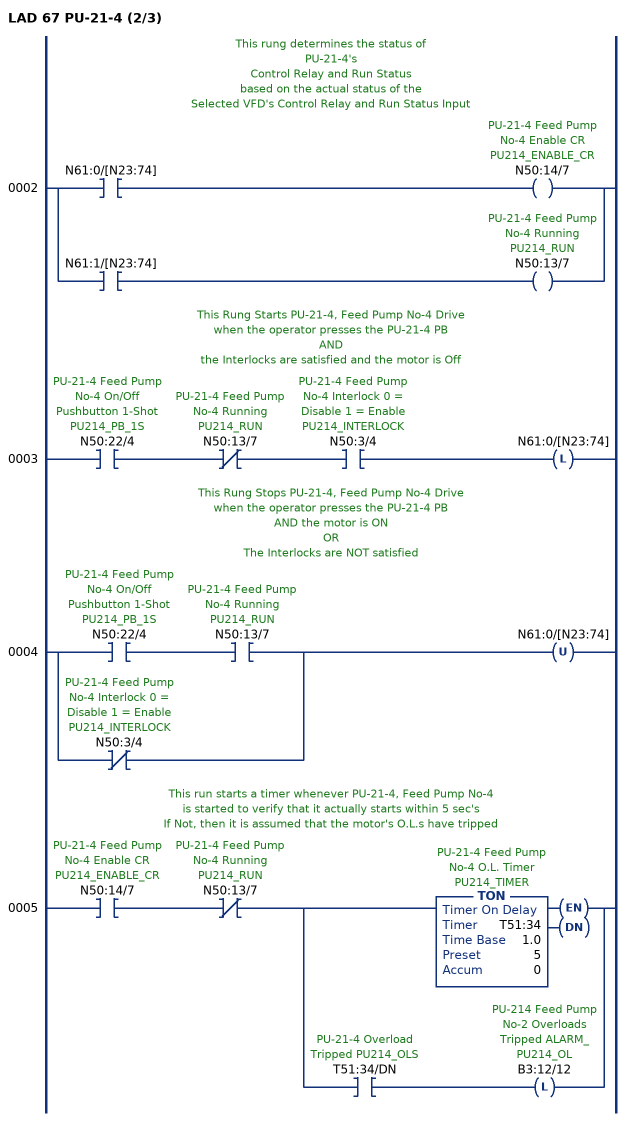
% Rung: 2 %
% This rung determines the status of
% PU-21-4's
% Control Relay and Run Status
% based on the actual status of the
% Selected VFD's Control Relay and Run Status Input %
SOR BST XIC N61:0/[N23:74] OTE N50:14/7 NXB XIC N61:1/[N23:74] OTE N50:13/7 BND EOR
%   N61:0  VFD_ENABLE_BITS  "These Bits Enable the appropriate VFD" %
%   N23:74  FIC214_OUT_PTR  "FIC-21-4 Feed Flow No-4 Output Pointer Determines which VFD is controled by FIC" %
%   N50:14/7  PU214_ENABLE_CR  "PU-21-4 Feed Pump No-4 Enable CR" %
%   N61:1  VFD_RUN_BITS_1  "These Bits Initcate the Status Off/Running for the appropriate VFD" %
%   N50:13/7  PU214_RUN  "PU-21-4 Feed Pump No-4 Running" %
% Rung: 3 %
% This Rung Starts PU-21-4, Feed Pump No-4 Drive
% when the operator presses the PU-21-4 PB
% AND
% the Interlocks are satisfied and the motor is Off %
SOR XIC N50:22/4 XIO N50:13/7 XIC N50:3/4 OTL N61:0/[N23:74] EOR
%   N50:22/4  PU214_PB_1S  "PU-21-4 Feed Pump No-4 On/Off Pushbutton 1-Shot" %
%   N50:13/7  PU214_RUN  "PU-21-4 Feed Pump No-4 Running" %
%   N50:3/4  PU214_INTERLOCK  "PU-21-4 Feed Pump No-4 Interlock 0 = Disable 1 = Enable" %
%   N61:0  VFD_ENABLE_BITS  "These Bits Enable the appropriate VFD" %
%   N23:74  FIC214_OUT_PTR  "FIC-21-4 Feed Flow No-4 Output Pointer Determines which VFD is controled by FIC" %
% Rung: 4 %
% This Rung Stops PU-21-4, Feed Pump No-4 Drive
% when the operator presses the PU-21-4 PB
% AND the motor is ON
% OR
% The Interlocks are NOT satisfied %
SOR BST XIC N50:22/4 XIC N50:13/7 NXB XIO N50:3/4 BND OTU N61:0/[N23:74] EOR
%   N50:22/4  PU214_PB_1S  "PU-21-4 Feed Pump No-4 On/Off Pushbutton 1-Shot" %
%   N50:13/7  PU214_RUN  "PU-21-4 Feed Pump No-4 Running" %
%   N50:3/4  PU214_INTERLOCK  "PU-21-4 Feed Pump No-4 Interlock 0 = Disable 1 = Enable" %
%   N61:0  VFD_ENABLE_BITS  "These Bits Enable the appropriate VFD" %
%   N23:74  FIC214_OUT_PTR  "FIC-21-4 Feed Flow No-4 Output Pointer Determines which VFD is controled by FIC" %
% Rung: 5 %
% This run starts a timer whenever PU-21-4, Feed Pump No-4
% is started to verify that it actually starts within 5 sec's
% If Not, then it is assumed that the motor's O.L.s have tripped %
SOR XIC N50:14/7 XIO N50:13/7 BST TON T51:34 1.0 5 0 NXB XIC T51:34/DN OTL B3:12/12 BND EOR
%   N50:14/7  PU214_ENABLE_CR  "PU-21-4 Feed Pump No-4 Enable CR" %
%   N50:13/7  PU214_RUN  "PU-21-4 Feed Pump No-4 Running" %
%   T51:34  PU214_TIMER  "PU-21-4 Feed Pump No-4 O.L. Timer" %
%   T51:34/DN  PU214_OLS  "PU-21-4 Overload Tripped" %
%   B3:12/12  ALARM_PU214_OL  "PU-214 Feed Pump No-2 Overloads Tripped" %

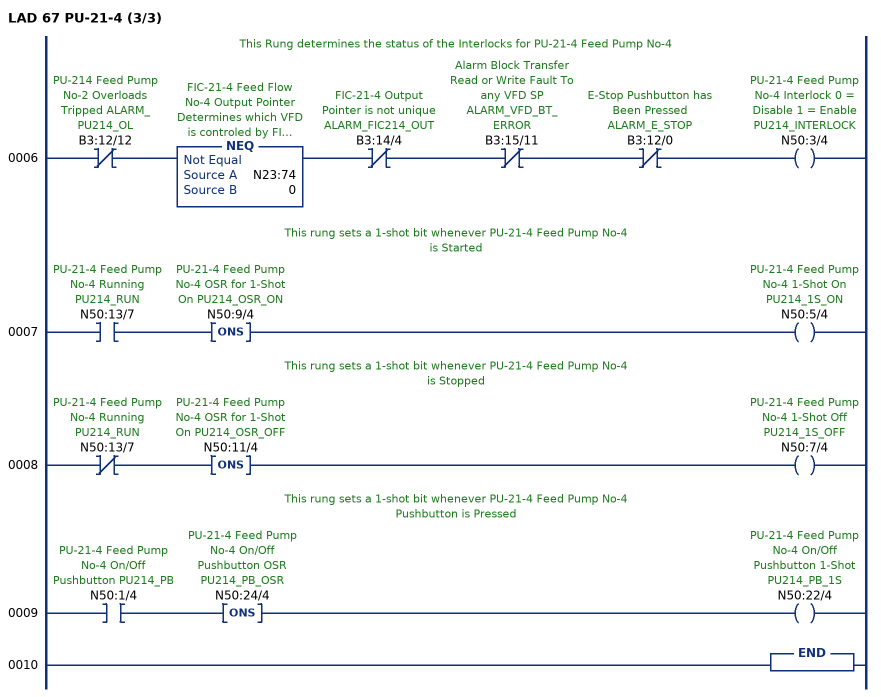
% Rung: 6 %
% This Rung determines the status of the Interlocks for PU-21-4 Feed Pump No-4 %
SOR XIO B3:12/12 NEQ N23:74 0 XIO B3:14/4 XIO B3:15/11 XIO B3:12/0 OTE N50:3/4 EOR
%   B3:12/12  ALARM_PU214_OL  "PU-214 Feed Pump No-2 Overloads Tripped" %
%   N23:74  FIC214_OUT_PTR  "FIC-21-4 Feed Flow No-4 Output Pointer Determines which VFD is controled by FIC" %
%   B3:14/4  ALARM_FIC214_OUT  "FIC-21-4 Output Pointer is not unique" %
%   B3:15/11  ALARM_VFD_BT_ERROR  "Alarm Block Transfer Read or Write Fault To any VFD SP" %
%   B3:12/0  ALARM_E_STOP  "E-Stop Pushbutton has Been Pressed" %
%   N50:3/4  PU214_INTERLOCK  "PU-21-4 Feed Pump No-4 Interlock 0 = Disable 1 = Enable" %
% Rung: 7 %
% This rung sets a 1-shot bit whenever PU-21-4 Feed Pump No-4
% is Started %
SOR XIC N50:13/7 OSR N50:9/4 OTE N50:5/4 EOR
%   N50:13/7  PU214_RUN  "PU-21-4 Feed Pump No-4 Running" %
%   N50:9/4  PU214_OSR_ON  "PU-21-4 Feed Pump No-4 OSR for 1-Shot On" %
%   N50:5/4  PU214_1S_ON  "PU-21-4 Feed Pump No-4 1-Shot On" %
% Rung: 8 %
% This rung sets a 1-shot bit whenever PU-21-4 Feed Pump No-4
% is Stopped %
SOR XIO N50:13/7 OSR N50:11/4 OTE N50:7/4 EOR
%   N50:13/7  PU214_RUN  "PU-21-4 Feed Pump No-4 Running" %
%   N50:11/4  PU214_OSR_OFF  "PU-21-4 Feed Pump No-4 OSR for 1-Shot On" %
%   N50:7/4  PU214_1S_OFF  "PU-21-4 Feed Pump No-4 1-Shot Off" %
% Rung: 9 %
% This rung sets a 1-shot bit whenever PU-21-4 Feed Pump No-4
% Pushbutton is Pressed %
SOR XIC N50:1/4 OSR N50:24/4 OTE N50:22/4 EOR
%   N50:1/4  PU214_PB  "PU-21-4 Feed Pump No-4 On/Off Pushbutton" %
%   N50:24/4  PU214_PB_OSR  "PU-21-4 Feed Pump No-4 On/Off Pushbutton OSR" %
%   N50:22/4  PU214_PB_1S  "PU-21-4 Feed Pump No-4 On/Off Pushbutton 1-Shot" %
% Rung: 10 %
SOR END EOR

LADDER 69 "PU-22-1"    % PU-22-1 Level Pump No-1 Controls %
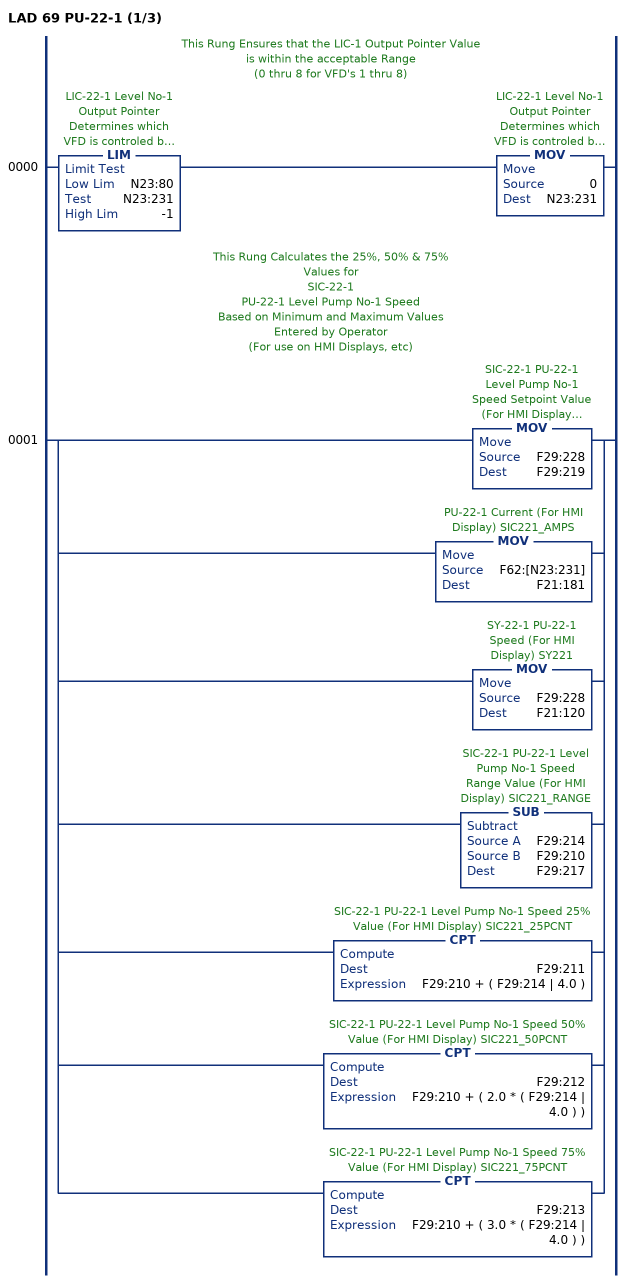
% Rung: 0 %
% This Rung Ensures that the LIC-1 Output Pointer Value
% is within the acceptable Range
% (0 thru 8 for VFD's 1 thru 8) %
SOR LIM N23:80 N23:231 -1 MOV 0 N23:231 EOR
%   N23:80  MAX_VFD_ALLOWED_1  "Maximum Number of VFDs Available Plus 1" %
%   N23:231  LIC221_OUT_PTR  "LIC-22-1 Level No-1 Output Pointer Determines which VFD is controled by LIC" %
% Rung: 1 %
% This Rung Calculates the 25%, 50% & 75%
% Values for
% SIC-22-1
% PU-22-1 Level Pump No-1 Speed
% Based on Minimum and Maximum Values
% Entered by Operator
% (For use on HMI Displays, etc) %
SOR BST MOV F29:228 F29:219 NXB MOV F62:[N23:231] F21:181 NXB MOV F29:228 F21:120 NXB SUB F29:214 F29:210 F29:217 NXB CPT F29:211 " F29:210 + ( F29:214 | 4.0 ) " NXB CPT F29:212 " F29:210 + ( 2.0 * ( F29:214 | 4.0 ) ) " NXB CPT F29:213 " F29:210 + ( 3.0 * ( F29:214 | 4.0 ) ) " BND EOR
%   F29:228  LIC221_OUT_FP  "LIC-22-1 Output Value (For HMI Display)" %
%   F29:219  SIC221_SP_FP  "SIC-22-1 PU-22-1 Level Pump No-1 Speed Setpoint Value (For HMI Display)" %
%   N23:231  LIC221_OUT_PTR  "LIC-22-1 Level No-1 Output Pointer Determines which VFD is controled by LIC" %
%   F21:181  SIC221_AMPS  "PU-22-1 Current (For HMI Display)" %
%   F21:120  SY221  "SY-22-1 PU-22-1 Speed (For HMI Display)" %
%   F29:214  SIC221_MAX  "SIC-22-1 PU-22-1 Level Pump No-1 Freq at 100% Value (For HMI Display)" %
%   F29:210  SIC221_MIN  "SIC-22-1 PU-22-1 Level Pump No-1 Speed 0% Value (For HMI Display)" %
%   F29:217  SIC221_RANGE  "SIC-22-1 PU-22-1 Level Pump No-1 Speed Range Value (For HMI Display)" %
%   F29:211  SIC221_25PCNT  "SIC-22-1 PU-22-1 Level Pump No-1 Speed 25% Value (For HMI Display)" %
%   F29:212  SIC221_50PCNT  "SIC-22-1 PU-22-1 Level Pump No-1 Speed 50% Value (For HMI Display)" %
%   F29:213  SIC221_75PCNT  "SIC-22-1 PU-22-1 Level Pump No-1 Speed 75% Value (For HMI Display)" %

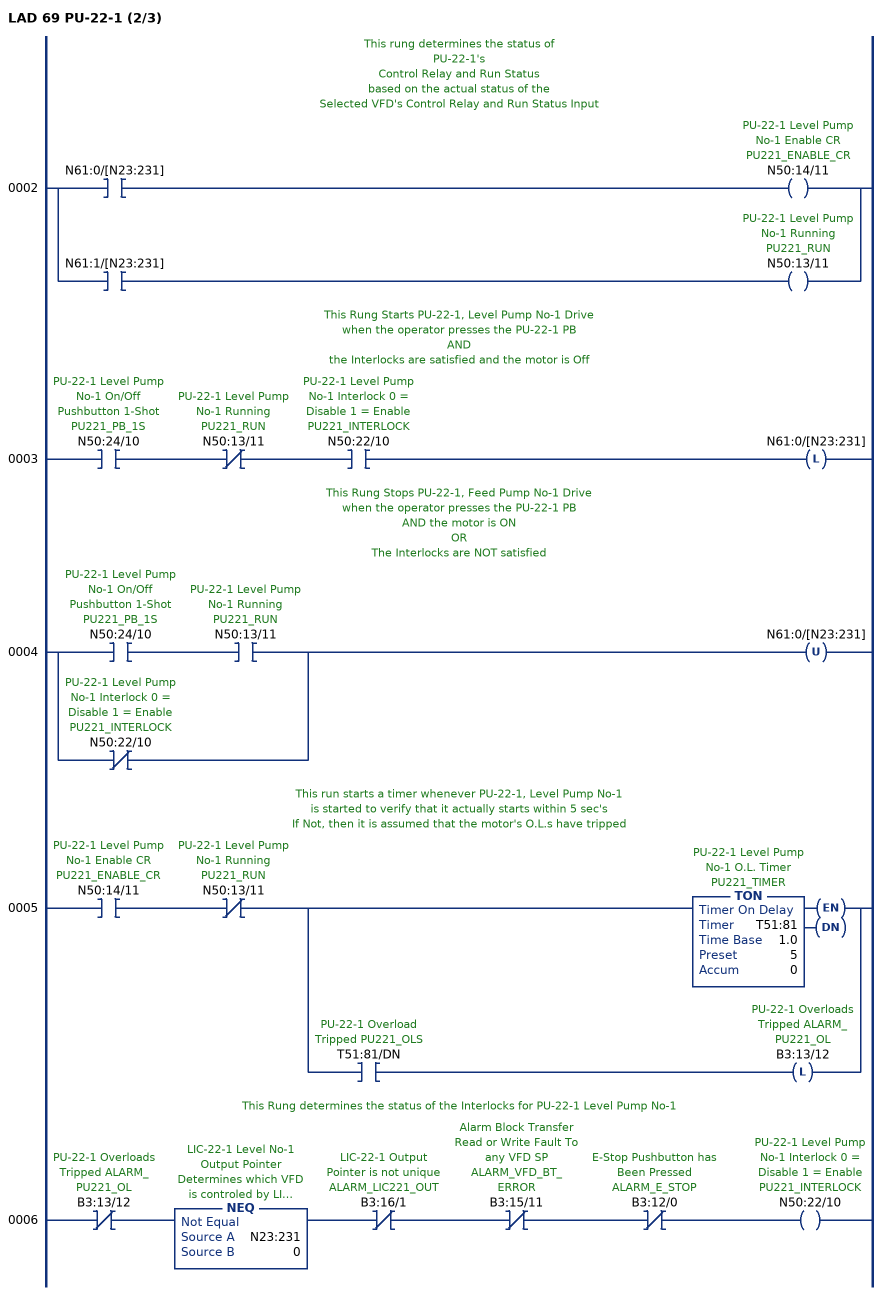
% Rung: 2 %
% This rung determines the status of
% PU-22-1's
% Control Relay and Run Status
% based on the actual status of the
% Selected VFD's Control Relay and Run Status Input %
SOR BST XIC N61:0/[N23:231] OTE N50:14/11 NXB XIC N61:1/[N23:231] OTE N50:13/11 BND EOR
%   N61:0  VFD_ENABLE_BITS  "These Bits Enable the appropriate VFD" %
%   N23:231  LIC221_OUT_PTR  "LIC-22-1 Level No-1 Output Pointer Determines which VFD is controled by LIC" %
%   N50:14/11  PU221_ENABLE_CR  "PU-22-1 Level Pump No-1 Enable CR" %
%   N61:1  VFD_RUN_BITS_1  "These Bits Initcate the Status Off/Running for the appropriate VFD" %
%   N50:13/11  PU221_RUN  "PU-22-1 Level Pump No-1 Running" %
% Rung: 3 %
% This Rung Starts PU-22-1, Level Pump No-1 Drive
% when the operator presses the PU-22-1 PB
% AND
% the Interlocks are satisfied and the motor is Off %
SOR XIC N50:24/10 XIO N50:13/11 XIC N50:22/10 OTL N61:0/[N23:231] EOR
%   N50:24/10  PU221_PB_1S  "PU-22-1 Level Pump No-1 On/Off Pushbutton 1-Shot" %
%   N50:13/11  PU221_RUN  "PU-22-1 Level Pump No-1 Running" %
%   N50:22/10  PU221_INTERLOCK  "PU-22-1 Level Pump No-1 Interlock 0 = Disable 1 = Enable" %
%   N61:0  VFD_ENABLE_BITS  "These Bits Enable the appropriate VFD" %
%   N23:231  LIC221_OUT_PTR  "LIC-22-1 Level No-1 Output Pointer Determines which VFD is controled by LIC" %
% Rung: 4 %
% This Rung Stops PU-22-1, Feed Pump No-1 Drive
% when the operator presses the PU-22-1 PB
% AND the motor is ON
% OR
% The Interlocks are NOT satisfied %
SOR BST XIC N50:24/10 XIC N50:13/11 NXB XIO N50:22/10 BND OTU N61:0/[N23:231] EOR
%   N50:24/10  PU221_PB_1S  "PU-22-1 Level Pump No-1 On/Off Pushbutton 1-Shot" %
%   N50:13/11  PU221_RUN  "PU-22-1 Level Pump No-1 Running" %
%   N50:22/10  PU221_INTERLOCK  "PU-22-1 Level Pump No-1 Interlock 0 = Disable 1 = Enable" %
%   N61:0  VFD_ENABLE_BITS  "These Bits Enable the appropriate VFD" %
%   N23:231  LIC221_OUT_PTR  "LIC-22-1 Level No-1 Output Pointer Determines which VFD is controled by LIC" %
% Rung: 5 %
% This run starts a timer whenever PU-22-1, Level Pump No-1
% is started to verify that it actually starts within 5 sec's
% If Not, then it is assumed that the motor's O.L.s have tripped %
SOR XIC N50:14/11 XIO N50:13/11 BST TON T51:81 1.0 5 0 NXB XIC T51:81/DN OTL B3:13/12 BND EOR
%   N50:14/11  PU221_ENABLE_CR  "PU-22-1 Level Pump No-1 Enable CR" %
%   N50:13/11  PU221_RUN  "PU-22-1 Level Pump No-1 Running" %
%   T51:81  PU221_TIMER  "PU-22-1 Level Pump No-1 O.L. Timer" %
%   T51:81/DN  PU221_OLS  "PU-22-1 Overload Tripped" %
%   B3:13/12  ALARM_PU221_OL  "PU-22-1 Overloads Tripped" %
% Rung: 6 %
% This Rung determines the status of the Interlocks for PU-22-1 Level Pump No-1 %
SOR XIO B3:13/12 NEQ N23:231 0 XIO B3:16/1 XIO B3:15/11 XIO B3:12/0 OTE N50:22/10 EOR
%   B3:13/12  ALARM_PU221_OL  "PU-22-1 Overloads Tripped" %
%   N23:231  LIC221_OUT_PTR  "LIC-22-1 Level No-1 Output Pointer Determines which VFD is controled by LIC" %
%   B3:16/1  ALARM_LIC221_OUT  "LIC-22-1 Output Pointer is not unique" %
%   B3:15/11  ALARM_VFD_BT_ERROR  "Alarm Block Transfer Read or Write Fault To any VFD SP" %
%   B3:12/0  ALARM_E_STOP  "E-Stop Pushbutton has Been Pressed" %
%   N50:22/10  PU221_INTERLOCK  "PU-22-1 Level Pump No-1 Interlock 0 = Disable 1 = Enable" %

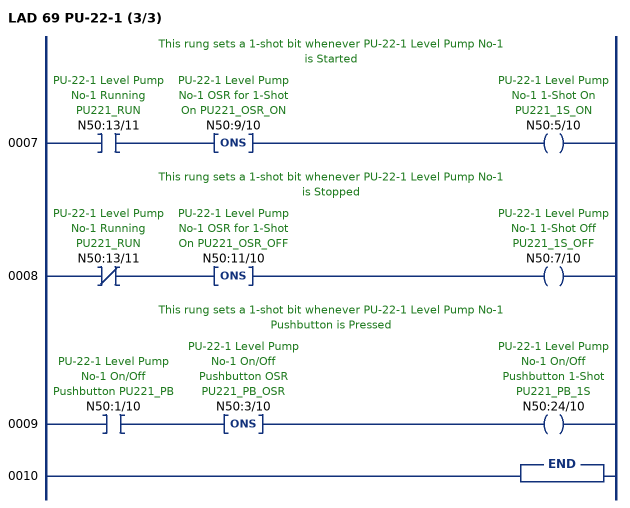
% Rung: 7 %
% This rung sets a 1-shot bit whenever PU-22-1 Level Pump No-1
% is Started %
SOR XIC N50:13/11 OSR N50:9/10 OTE N50:5/10 EOR
%   N50:13/11  PU221_RUN  "PU-22-1 Level Pump No-1 Running" %
%   N50:9/10  PU221_OSR_ON  "PU-22-1 Level Pump No-1 OSR for 1-Shot On" %
%   N50:5/10  PU221_1S_ON  "PU-22-1 Level Pump No-1 1-Shot On" %
% Rung: 8 %
% This rung sets a 1-shot bit whenever PU-22-1 Level Pump No-1
% is Stopped %
SOR XIO N50:13/11 OSR N50:11/10 OTE N50:7/10 EOR
%   N50:13/11  PU221_RUN  "PU-22-1 Level Pump No-1 Running" %
%   N50:11/10  PU221_OSR_OFF  "PU-22-1 Level Pump No-1 OSR for 1-Shot On" %
%   N50:7/10  PU221_1S_OFF  "PU-22-1 Level Pump No-1 1-Shot Off" %
% Rung: 9 %
% This rung sets a 1-shot bit whenever PU-22-1 Level Pump No-1
% Pushbutton is Pressed %
SOR XIC N50:1/10 OSR N50:3/10 OTE N50:24/10 EOR
%   N50:1/10  PU221_PB  "PU-22-1 Level Pump No-1 On/Off Pushbutton" %
%   N50:3/10  PU221_PB_OSR  "PU-22-1 Level Pump No-1 On/Off Pushbutton OSR" %
%   N50:24/10  PU221_PB_1S  "PU-22-1 Level Pump No-1 On/Off Pushbutton 1-Shot" %
% Rung: 10 %
SOR END EOR

LADDER 71 "PU-23"    % PU-23 Hot Oil Circ Pump Controls %
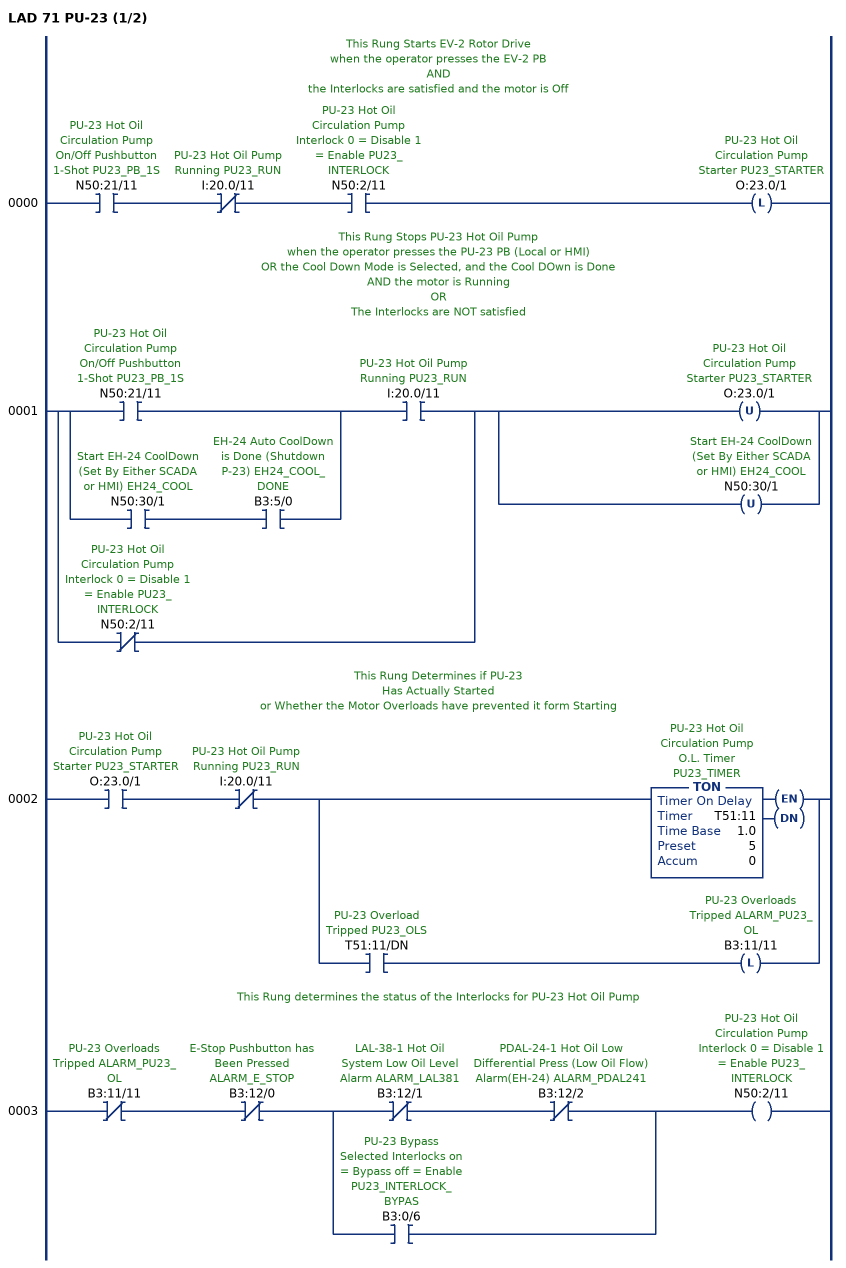
% Rung: 0 %
% This Rung Starts EV-2 Rotor Drive
% when the operator presses the EV-2 PB
% AND
% the Interlocks are satisfied and the motor is Off %
SOR XIC N50:21/11 XIO I:20.0/11 XIC N50:2/11 OTL O:23.0/1 EOR
%   N50:21/11  PU23_PB_1S  "PU-23 Hot Oil Circulation Pump On/Off Pushbutton 1-Shot" %
%   I:20.0/11  PU23_RUN  "PU-23 Hot Oil Pump Running" %
%   N50:2/11  PU23_INTERLOCK  "PU-23 Hot Oil Circulation Pump Interlock 0 = Disable 1 = Enable" %
%   O:23.0/1  PU23_STARTER  "PU-23 Hot Oil Circulation Pump Starter" %
% Rung: 1 %
% This Rung Stops PU-23 Hot Oil Pump
% when the operator presses the PU-23 PB (Local or HMI)
% OR the Cool Down Mode is Selected, and the Cool DOwn is Done
% AND the motor is Running
% OR
% The Interlocks are NOT satisfied %
SOR BST BST XIC N50:21/11 NXB XIC N50:30/1 XIC B3:5/0 BND XIC I:20.0/11 NXB XIO N50:2/11 BND BST OTU O:23.0/1 NXB OTU N50:30/1 BND EOR
%   N50:21/11  PU23_PB_1S  "PU-23 Hot Oil Circulation Pump On/Off Pushbutton 1-Shot" %
%   N50:30/1  EH24_COOL  "Start EH-24 CoolDown (Set By Either SCADA or HMI)" %
%   B3:5/0  EH24_COOL_DONE  "EH-24 Auto CoolDown is Done (Shutdown P-23)" %
%   I:20.0/11  PU23_RUN  "PU-23 Hot Oil Pump Running" %
%   N50:2/11  PU23_INTERLOCK  "PU-23 Hot Oil Circulation Pump Interlock 0 = Disable 1 = Enable" %
%   O:23.0/1  PU23_STARTER  "PU-23 Hot Oil Circulation Pump Starter" %
% Rung: 2 %
% This Rung Determines if PU-23
% Has Actually Started
% or Whether the Motor Overloads have prevented it form Starting %
SOR XIC O:23.0/1 XIO I:20.0/11 BST TON T51:11 1.0 5 0 NXB XIC T51:11/DN OTL B3:11/11 BND EOR
%   O:23.0/1  PU23_STARTER  "PU-23 Hot Oil Circulation Pump Starter" %
%   I:20.0/11  PU23_RUN  "PU-23 Hot Oil Pump Running" %
%   T51:11  PU23_TIMER  "PU-23 Hot Oil Circulation Pump O.L. Timer" %
%   T51:11/DN  PU23_OLS  "PU-23 Overload Tripped" %
%   B3:11/11  ALARM_PU23_OL  "PU-23 Overloads Tripped" %
% Rung: 3 %
% This Rung determines the status of the Interlocks for PU-23 Hot Oil Pump %
SOR XIO B3:11/11 XIO B3:12/0 BST XIO B3:12/1 XIO B3:12/2 NXB XIC B3:0/6 BND OTE N50:2/11 EOR
%   B3:11/11  ALARM_PU23_OL  "PU-23 Overloads Tripped" %
%   B3:12/0  ALARM_E_STOP  "E-Stop Pushbutton has Been Pressed" %
%   B3:12/1  ALARM_LAL381  "LAL-38-1 Hot Oil System Low Oil Level Alarm" %
%   B3:12/2  ALARM_PDAL241  "PDAL-24-1 Hot Oil Low Differential Press (Low Oil Flow) Alarm(EH-24)" %
%   B3:0/6  PU23_INTERLOCK_BYPAS  "PU-23 Bypass Selected Interlocks on = Bypass off = Enable" %
%   N50:2/11  PU23_INTERLOCK  "PU-23 Hot Oil Circulation Pump Interlock 0 = Disable 1 = Enable" %

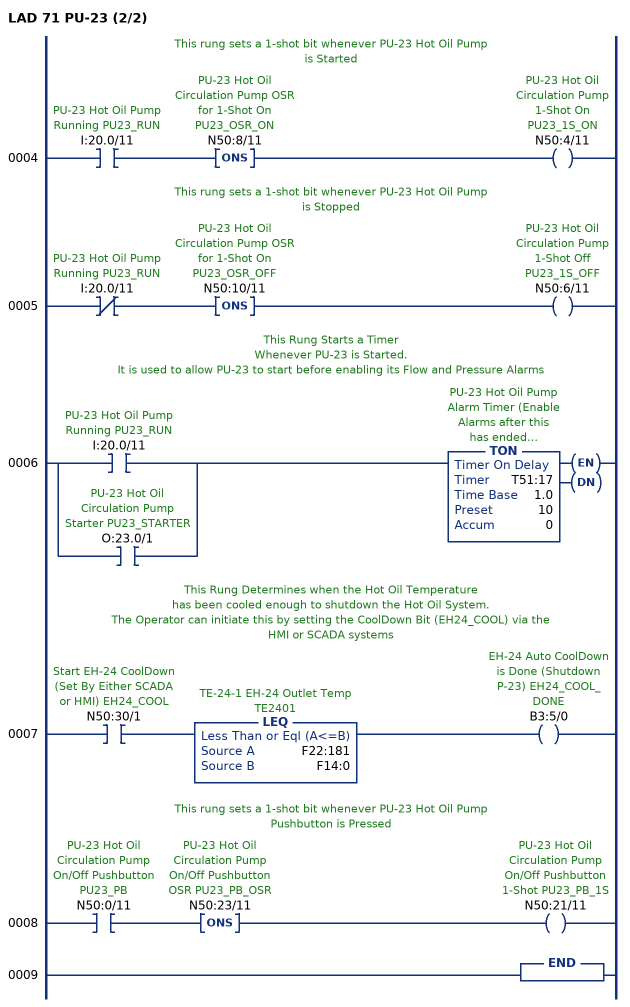
% Rung: 4 %
% This rung sets a 1-shot bit whenever PU-23 Hot Oil Pump
% is Started %
SOR XIC I:20.0/11 OSR N50:8/11 OTE N50:4/11 EOR
%   I:20.0/11  PU23_RUN  "PU-23 Hot Oil Pump Running" %
%   N50:8/11  PU23_OSR_ON  "PU-23 Hot Oil Circulation Pump OSR for 1-Shot On" %
%   N50:4/11  PU23_1S_ON  "PU-23 Hot Oil Circulation Pump 1-Shot On" %
% Rung: 5 %
% This rung sets a 1-shot bit whenever PU-23 Hot Oil Pump
% is Stopped %
SOR XIO I:20.0/11 OSR N50:10/11 OTE N50:6/11 EOR
%   I:20.0/11  PU23_RUN  "PU-23 Hot Oil Pump Running" %
%   N50:10/11  PU23_OSR_OFF  "PU-23 Hot Oil Circulation Pump OSR for 1-Shot On" %
%   N50:6/11  PU23_1S_OFF  "PU-23 Hot Oil Circulation Pump 1-Shot Off" %
% Rung: 6 %
% This Rung Starts a Timer
% Whenever PU-23 is Started.
% It is used to allow PU-23 to start before enabling its Flow and Pressure Alarms %
SOR BST XIC I:20.0/11 NXB XIC O:23.0/1 BND TON T51:17 1.0 10 0 EOR
%   I:20.0/11  PU23_RUN  "PU-23 Hot Oil Pump Running" %
%   O:23.0/1  PU23_STARTER  "PU-23 Hot Oil Circulation Pump Starter" %
%   T51:17  PU23_ALARM_TMR  "PU-23 Hot Oil Pump Alarm Timer (Enable Alarms after this has ended)" %
% Rung: 7 %
% This Rung Determines when the Hot Oil Temperature
% has been cooled enough to shutdown the Hot Oil System.
% The Operator can initiate this by setting the CoolDown Bit (EH24_COOL) via the
% HMI or SCADA systems %
SOR XIC N50:30/1 LEQ F22:181 F14:0 OTE B3:5/0 EOR
%   N50:30/1  EH24_COOL  "Start EH-24 CoolDown (Set By Either SCADA or HMI)" %
%   F22:181  TE2401  "TE-24-1 EH-24 Outlet Temp" %
%   F14:0  EH24_COOLDOWN_SP  "EH-24 CoolDown Setpoint" %
%   B3:5/0  EH24_COOL_DONE  "EH-24 Auto CoolDown is Done (Shutdown P-23)" %
% Rung: 8 %
% This rung sets a 1-shot bit whenever PU-23 Hot Oil Pump
% Pushbutton is Pressed %
SOR XIC N50:0/11 OSR N50:23/11 OTE N50:21/11 EOR
%   N50:0/11  PU23_PB  "PU-23 Hot Oil Circulation Pump On/Off Pushbutton" %
%   N50:23/11  PU23_PB_OSR  "PU-23 Hot Oil Circulation Pump On/Off Pushbutton OSR" %
%   N50:21/11  PU23_PB_1S  "PU-23 Hot Oil Circulation Pump On/Off Pushbutton 1-Shot" %
% Rung: 9 %
SOR END EOR

LADDER 72 "EH-24"    % EH-24 Hot Oil Heater Controls %
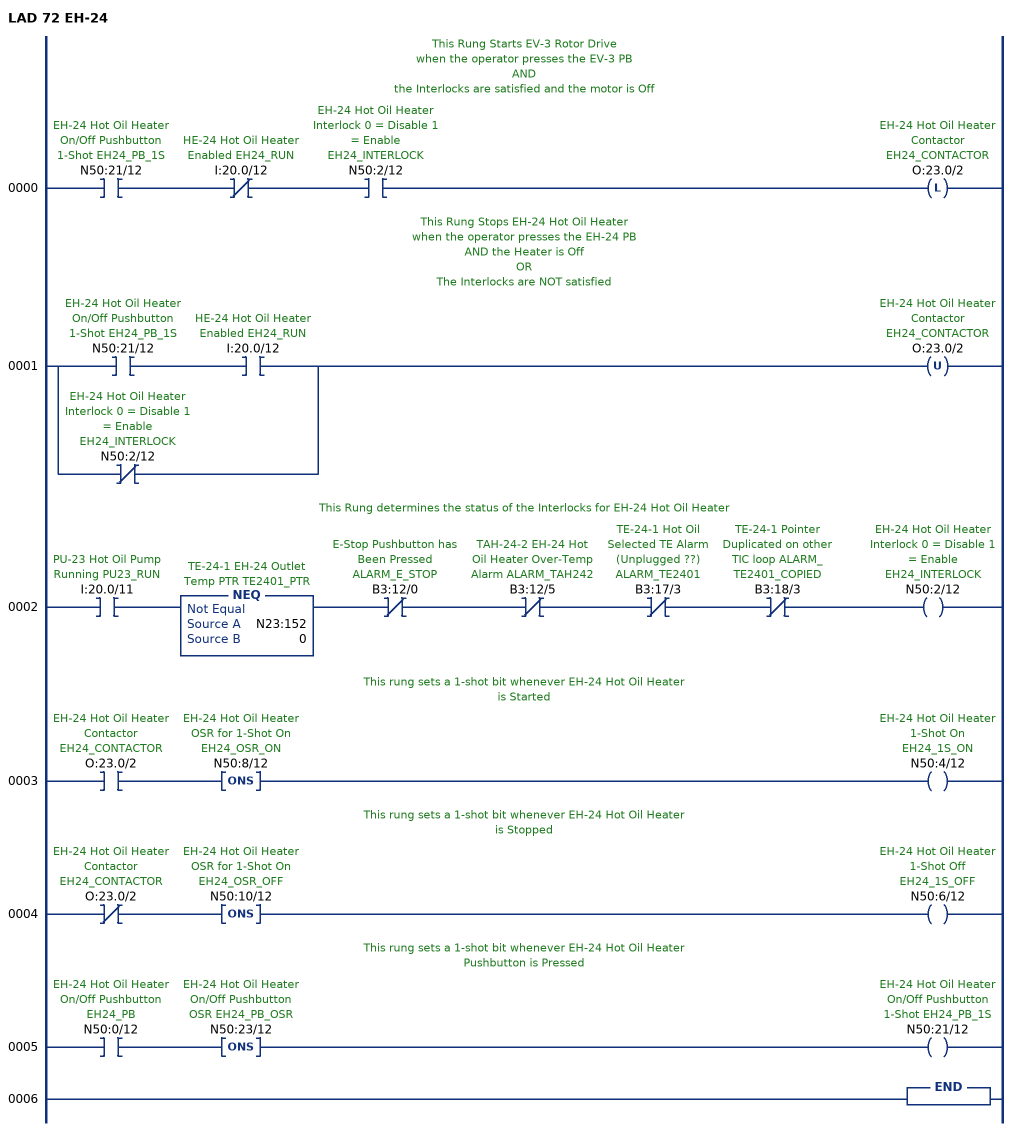
% Rung: 0 %
% This Rung Starts EV-3 Rotor Drive
% when the operator presses the EV-3 PB
% AND
% the Interlocks are satisfied and the motor is Off %
SOR XIC N50:21/12 XIO I:20.0/12 XIC N50:2/12 OTL O:23.0/2 EOR
%   N50:21/12  EH24_PB_1S  "EH-24 Hot Oil Heater On/Off Pushbutton 1-Shot" %
%   I:20.0/12  EH24_RUN  "HE-24 Hot Oil Heater Enabled" %
%   N50:2/12  EH24_INTERLOCK  "EH-24 Hot Oil Heater Interlock 0 = Disable 1 = Enable" %
%   O:23.0/2  EH24_CONTACTOR  "EH-24 Hot Oil Heater Contactor" %
% Rung: 1 %
% This Rung Stops EH-24 Hot Oil Heater
% when the operator presses the EH-24 PB
% AND the Heater is Off
% OR
% The Interlocks are NOT satisfied %
SOR BST XIC N50:21/12 XIC I:20.0/12 NXB XIO N50:2/12 BND OTU O:23.0/2 EOR
%   N50:21/12  EH24_PB_1S  "EH-24 Hot Oil Heater On/Off Pushbutton 1-Shot" %
%   I:20.0/12  EH24_RUN  "HE-24 Hot Oil Heater Enabled" %
%   N50:2/12  EH24_INTERLOCK  "EH-24 Hot Oil Heater Interlock 0 = Disable 1 = Enable" %
%   O:23.0/2  EH24_CONTACTOR  "EH-24 Hot Oil Heater Contactor" %
% Rung: 2 %
% This Rung determines the status of the Interlocks for EH-24 Hot Oil Heater %
SOR XIC I:20.0/11 NEQ N23:152 0 XIO B3:12/0 XIO B3:12/5 XIO B3:17/3 XIO B3:18/3 OTE N50:2/12 EOR
%   I:20.0/11  PU23_RUN  "PU-23 Hot Oil Pump Running" %
%   N23:152  TE2401_PTR  "TE-24-1 EH-24 Outlet Temp PTR" %
%   B3:12/0  ALARM_E_STOP  "E-Stop Pushbutton has Been Pressed" %
%   B3:12/5  ALARM_TAH242  "TAH-24-2 EH-24 Hot Oil Heater Over-Temp Alarm" %
%   B3:17/3  ALARM_TE2401  "TE-24-1 Hot Oil Selected TE Alarm (Unplugged ??)" %
%   B3:18/3  ALARM_TE2401_COPIED  "TE-24-1 Pointer Duplicated on other TIC loop" %
%   N50:2/12  EH24_INTERLOCK  "EH-24 Hot Oil Heater Interlock 0 = Disable 1 = Enable" %
% Rung: 3 %
% This rung sets a 1-shot bit whenever EH-24 Hot Oil Heater
% is Started %
SOR XIC O:23.0/2 OSR N50:8/12 OTE N50:4/12 EOR
%   O:23.0/2  EH24_CONTACTOR  "EH-24 Hot Oil Heater Contactor" %
%   N50:8/12  EH24_OSR_ON  "EH-24 Hot Oil Heater OSR for 1-Shot On" %
%   N50:4/12  EH24_1S_ON  "EH-24 Hot Oil Heater 1-Shot On" %
% Rung: 4 %
% This rung sets a 1-shot bit whenever EH-24 Hot Oil Heater
% is Stopped %
SOR XIO O:23.0/2 OSR N50:10/12 OTE N50:6/12 EOR
%   O:23.0/2  EH24_CONTACTOR  "EH-24 Hot Oil Heater Contactor" %
%   N50:10/12  EH24_OSR_OFF  "EH-24 Hot Oil Heater OSR for 1-Shot On" %
%   N50:6/12  EH24_1S_OFF  "EH-24 Hot Oil Heater 1-Shot Off" %
% Rung: 5 %
% This rung sets a 1-shot bit whenever EH-24 Hot Oil Heater
% Pushbutton is Pressed %
SOR XIC N50:0/12 OSR N50:23/12 OTE N50:21/12 EOR
%   N50:0/12  EH24_PB  "EH-24 Hot Oil Heater On/Off Pushbutton" %
%   N50:23/12  EH24_PB_OSR  "EH-24 Hot Oil Heater On/Off Pushbutton OSR" %
%   N50:21/12  EH24_PB_1S  "EH-24 Hot Oil Heater On/Off Pushbutton 1-Shot" %
% Rung: 6 %
SOR END EOR

LADDER 73 "VB-26"    % VB-26 Beach-Ross Vacuum Blower Controls %
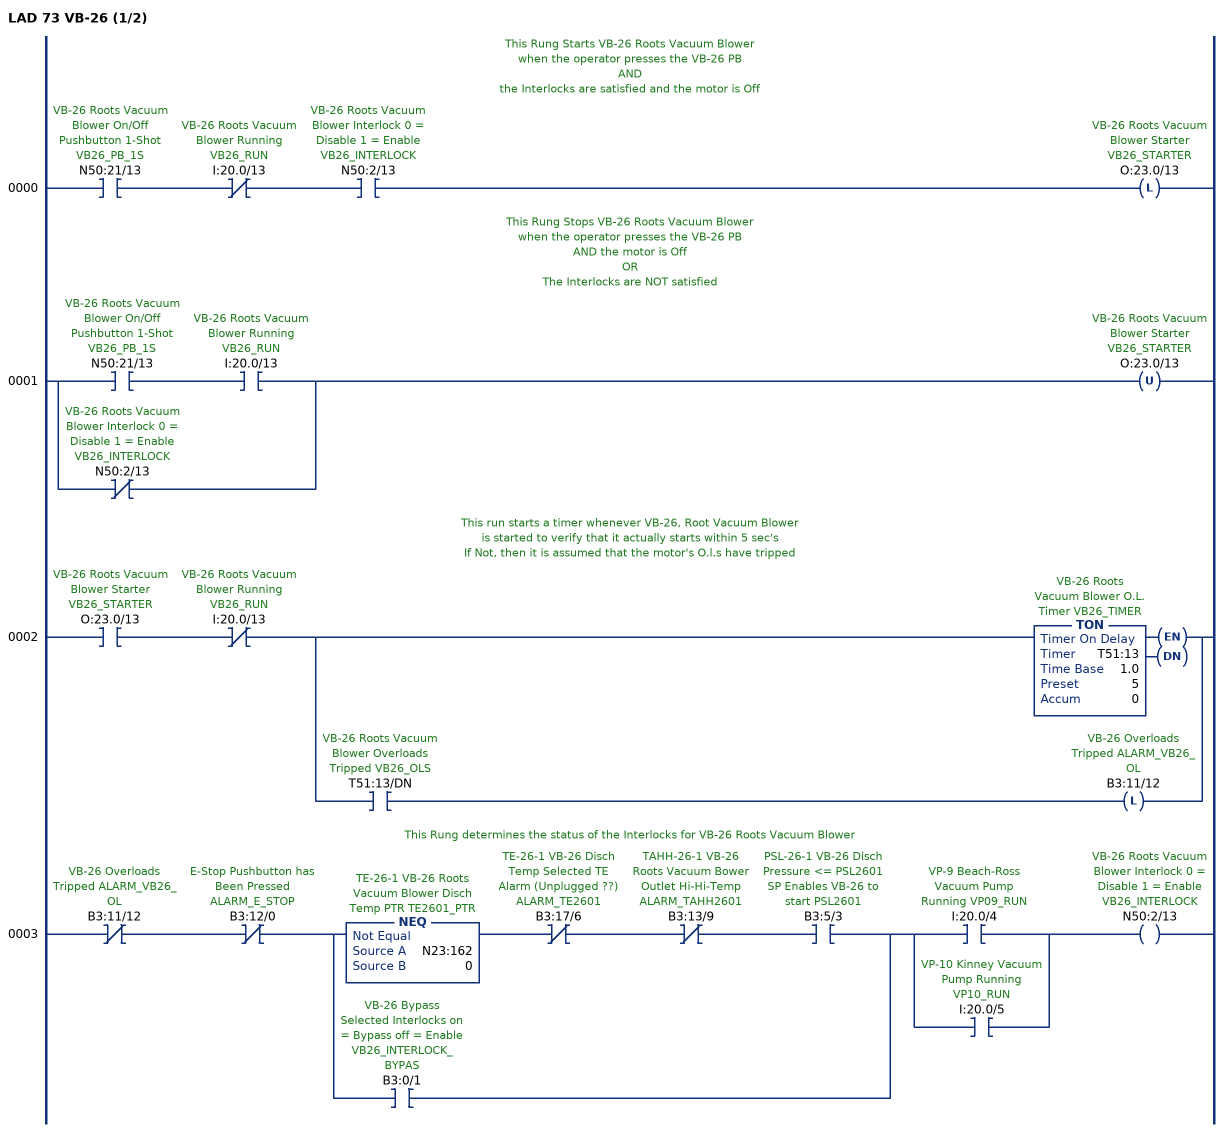
% Rung: 0 %
% This Rung Starts VB-26 Roots Vacuum Blower
% when the operator presses the VB-26 PB
% AND
% the Interlocks are satisfied and the motor is Off %
SOR XIC N50:21/13 XIO I:20.0/13 XIC N50:2/13 OTL O:23.0/13 EOR
%   N50:21/13  VB26_PB_1S  "VB-26 Roots Vacuum Blower On/Off Pushbutton 1-Shot" %
%   I:20.0/13  VB26_RUN  "VB-26 Roots Vacuum Blower Running" %
%   N50:2/13  VB26_INTERLOCK  "VB-26 Roots Vacuum Blower Interlock 0 = Disable 1 = Enable" %
%   O:23.0/13  VB26_STARTER  "VB-26 Roots Vacuum Blower Starter" %
% Rung: 1 %
% This Rung Stops VB-26 Roots Vacuum Blower
% when the operator presses the VB-26 PB
% AND the motor is Off
% OR
% The Interlocks are NOT satisfied %
SOR BST XIC N50:21/13 XIC I:20.0/13 NXB XIO N50:2/13 BND OTU O:23.0/13 EOR
%   N50:21/13  VB26_PB_1S  "VB-26 Roots Vacuum Blower On/Off Pushbutton 1-Shot" %
%   I:20.0/13  VB26_RUN  "VB-26 Roots Vacuum Blower Running" %
%   N50:2/13  VB26_INTERLOCK  "VB-26 Roots Vacuum Blower Interlock 0 = Disable 1 = Enable" %
%   O:23.0/13  VB26_STARTER  "VB-26 Roots Vacuum Blower Starter" %
% Rung: 2 %
% This run starts a timer whenever VB-26, Root Vacuum Blower
% is started to verify that it actually starts within 5 sec's
% If Not, then it is assumed that the motor's O.l.s have tripped %
SOR XIC O:23.0/13 XIO I:20.0/13 BST TON T51:13 1.0 5 0 NXB XIC T51:13/DN OTL B3:11/12 BND EOR
%   O:23.0/13  VB26_STARTER  "VB-26 Roots Vacuum Blower Starter" %
%   I:20.0/13  VB26_RUN  "VB-26 Roots Vacuum Blower Running" %
%   T51:13  VB26_TIMER  "VB-26 Roots Vacuum Blower O.L. Timer" %
%   T51:13/DN  VB26_OLS  "VB-26 Roots Vacuum Blower Overloads Tripped" %
%   B3:11/12  ALARM_VB26_OL  "VB-26 Overloads Tripped" %
% Rung: 3 %
% This Rung determines the status of the Interlocks for VB-26 Roots Vacuum Blower %
SOR XIO B3:11/12 XIO B3:12/0 BST NEQ N23:162 0 XIO B3:17/6 XIO B3:13/9 XIC B3:5/3 NXB XIC B3:0/1 BND BST XIC I:20.0/4 NXB XIC I:20.0/5 BND OTE N50:2/13 EOR
%   B3:11/12  ALARM_VB26_OL  "VB-26 Overloads Tripped" %
%   B3:12/0  ALARM_E_STOP  "E-Stop Pushbutton has Been Pressed" %
%   N23:162  TE2601_PTR  "TE-26-1 VB-26 Roots Vacuum Blower Disch Temp PTR" %
%   B3:17/6  ALARM_TE2601  "TE-26-1 VB-26 Disch Temp Selected TE Alarm (Unplugged ??)" %
%   B3:13/9  ALARM_TAHH2601  "TAHH-26-1 VB-26 Roots Vacuum Bower Outlet Hi-Hi-Temp" %
%   B3:5/3  PSL2601  "PSL-26-1 VB-26 Disch Pressure <= PSL2601 SP Enables VB-26 to start" %
%   B3:0/1  VB26_INTERLOCK_BYPAS  "VB-26 Bypass Selected Interlocks on = Bypass off = Enable" %
%   I:20.0/4  VP09_RUN  "VP-9 Beach-Ross Vacuum Pump Running" %
%   I:20.0/5  VP10_RUN  "VP-10 Kinney Vacuum Pump Running" %
%   N50:2/13  VB26_INTERLOCK  "VB-26 Roots Vacuum Blower Interlock 0 = Disable 1 = Enable" %

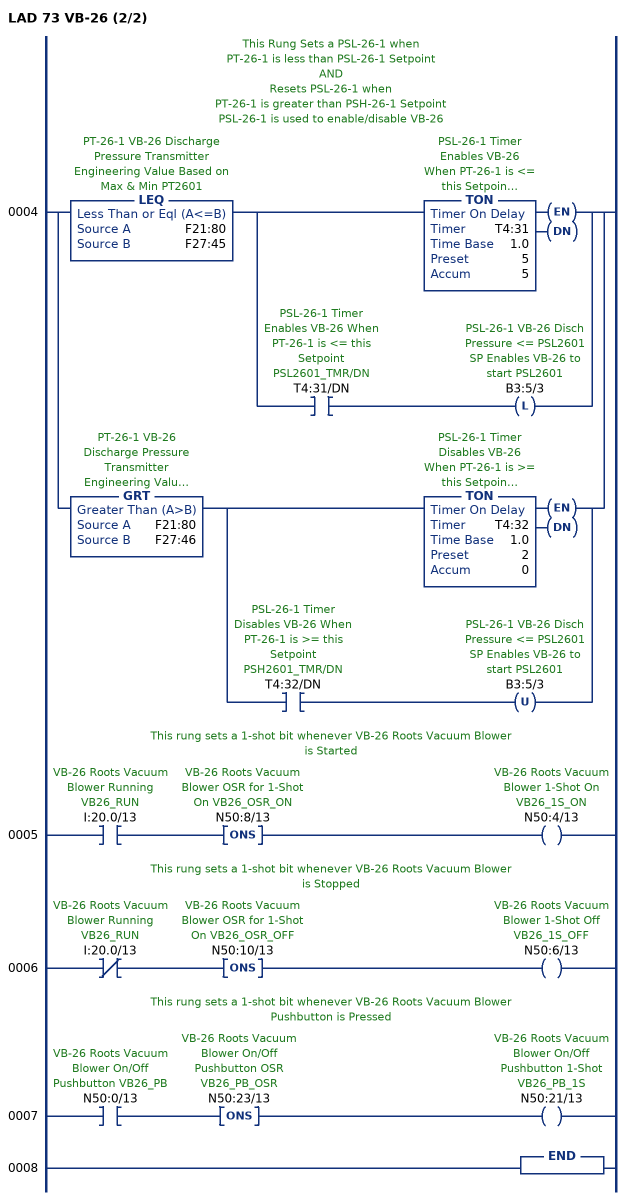
% Rung: 4 %
% This Rung Sets a PSL-26-1 when
% PT-26-1 is less than PSL-26-1 Setpoint
% AND
% Resets PSL-26-1 when
% PT-26-1 is greater than PSH-26-1 Setpoint
% 
% PSL-26-1 is used to enable/disable VB-26 %
SOR BST LEQ F21:80 F27:45 BST TON T4:31 1.0 5 5 NXB XIC T4:31/DN OTL B3:5/3 BND NXB GRT F21:80 F27:46 BST TON T4:32 1.0 2 0 NXB XIC T4:32/DN OTU B3:5/3 BND BND EOR
%   F21:80  PT2601  "PT-26-1 VB-26 Discharge Pressure Transmitter Engineering Value Based on Max & Min" %
%   F27:45  PSL2601_SP  "PSL-26-1 Setpoint Enables VB-26 When PT-26-1 is LESS than this value" %
%   T4:31  PSL2601_TMR  "PSL-26-1 Timer Enables VB-26 When PT-26-1 is <= this Setpoint" %
%   B3:5/3  PSL2601  "PSL-26-1 VB-26 Disch Pressure <= PSL2601 SP Enables VB-26 to start" %
%   F27:46  PSH2601_SP  "PSL-26-1 Setpoint Disables VB-26 When PT-26-1 is >= than this value" %
%   T4:32  PSH2601_TMR  "PSL-26-1 Timer Disables VB-26 When PT-26-1 is >= this Setpoint" %
% Rung: 5 %
% This rung sets a 1-shot bit whenever VB-26 Roots Vacuum Blower
% is Started %
SOR XIC I:20.0/13 OSR N50:8/13 OTE N50:4/13 EOR
%   I:20.0/13  VB26_RUN  "VB-26 Roots Vacuum Blower Running" %
%   N50:8/13  VB26_OSR_ON  "VB-26 Roots Vacuum Blower OSR for 1-Shot On" %
%   N50:4/13  VB26_1S_ON  "VB-26 Roots Vacuum Blower 1-Shot On" %
% Rung: 6 %
% This rung sets a 1-shot bit whenever VB-26 Roots Vacuum Blower
% is Stopped %
SOR XIO I:20.0/13 OSR N50:10/13 OTE N50:6/13 EOR
%   I:20.0/13  VB26_RUN  "VB-26 Roots Vacuum Blower Running" %
%   N50:10/13  VB26_OSR_OFF  "VB-26 Roots Vacuum Blower OSR for 1-Shot On" %
%   N50:6/13  VB26_1S_OFF  "VB-26 Roots Vacuum Blower 1-Shot Off" %
% Rung: 7 %
% This rung sets a 1-shot bit whenever VB-26 Roots Vacuum Blower
% Pushbutton is Pressed %
SOR XIC N50:0/13 OSR N50:23/13 OTE N50:21/13 EOR
%   N50:0/13  VB26_PB  "VB-26 Roots Vacuum Blower On/Off Pushbutton" %
%   N50:23/13  VB26_PB_OSR  "VB-26 Roots Vacuum Blower On/Off Pushbutton OSR" %
%   N50:21/13  VB26_PB_1S  "VB-26 Roots Vacuum Blower On/Off Pushbutton 1-Shot" %
% Rung: 8 %
SOR END EOR

LADDER 74 "PU-30"    % PU-30 Cooling Water Header Booster Pump Controls %
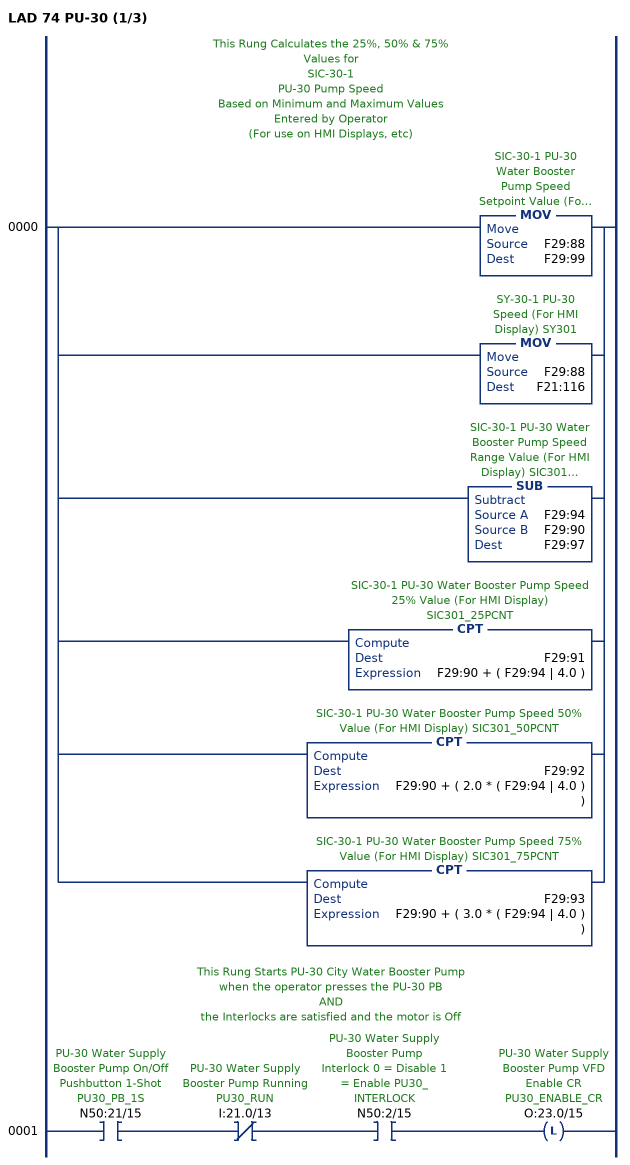
% Rung: 0 %
% This Rung Calculates the 25%, 50% & 75%
% Values for
% SIC-30-1
% PU-30 Pump Speed
% Based on Minimum and Maximum Values
% Entered by Operator
% (For use on HMI Displays, etc) %
SOR BST MOV F29:88 F29:99 NXB MOV F29:88 F21:116 NXB SUB F29:94 F29:90 F29:97 NXB CPT F29:91 " F29:90 + ( F29:94 | 4.0 ) " NXB CPT F29:92 " F29:90 + ( 2.0 * ( F29:94 | 4.0 ) ) " NXB CPT F29:93 " F29:90 + ( 3.0 * ( F29:94 | 4.0 ) ) " BND EOR
%   F29:88  PIC301_OUT_FP  "PIC-30-1 Output Value (For HMI Display)" %
%   F29:99  SIC301_SP_FP  "SIC-30-1 PU-30 Water Booster Pump Speed Setpoint Value (For HMI Display)" %
%   F21:116  SY301  "SY-30-1 PU-30 Speed (For HMI Display)" %
%   F29:94  SIC301_MAX  "SIC-30-1 PU-30 Water Booster Pump Speed 100% Value (For HMI Display)" %
%   F29:90  SIC301_MIN  "SIC-30-1 PU-30 Water Booster Pump Speed 0% Value (For HMI Display)" %
%   F29:97  SIC301_RANGE  "SIC-30-1 PU-30 Water Booster Pump Speed Range Value (For HMI Display)" %
%   F29:91  SIC301_25PCNT  "SIC-30-1 PU-30 Water Booster Pump Speed 25% Value (For HMI Display)" %
%   F29:92  SIC301_50PCNT  "SIC-30-1 PU-30 Water Booster Pump Speed 50% Value (For HMI Display)" %
%   F29:93  SIC301_75PCNT  "SIC-30-1 PU-30 Water Booster Pump Speed 75% Value (For HMI Display)" %
% Rung: 1 %
% This Rung Starts PU-30 City Water Booster Pump
% when the operator presses the PU-30 PB
% AND
% the Interlocks are satisfied and the motor is Off %
SOR XIC N50:21/15 XIO I:21.0/13 XIC N50:2/15 OTL O:23.0/15 EOR
%   N50:21/15  PU30_PB_1S  "PU-30 Water Supply Booster Pump On/Off Pushbutton 1-Shot" %
%   I:21.0/13  PU30_RUN  "PU-30 Water Supply Booster Pump Running" %
%   N50:2/15  PU30_INTERLOCK  "PU-30 Water Supply Booster Pump Interlock 0 = Disable 1 = Enable" %
%   O:23.0/15  PU30_ENABLE_CR  "PU-30 Water Supply Booster Pump VFD Enable CR" %

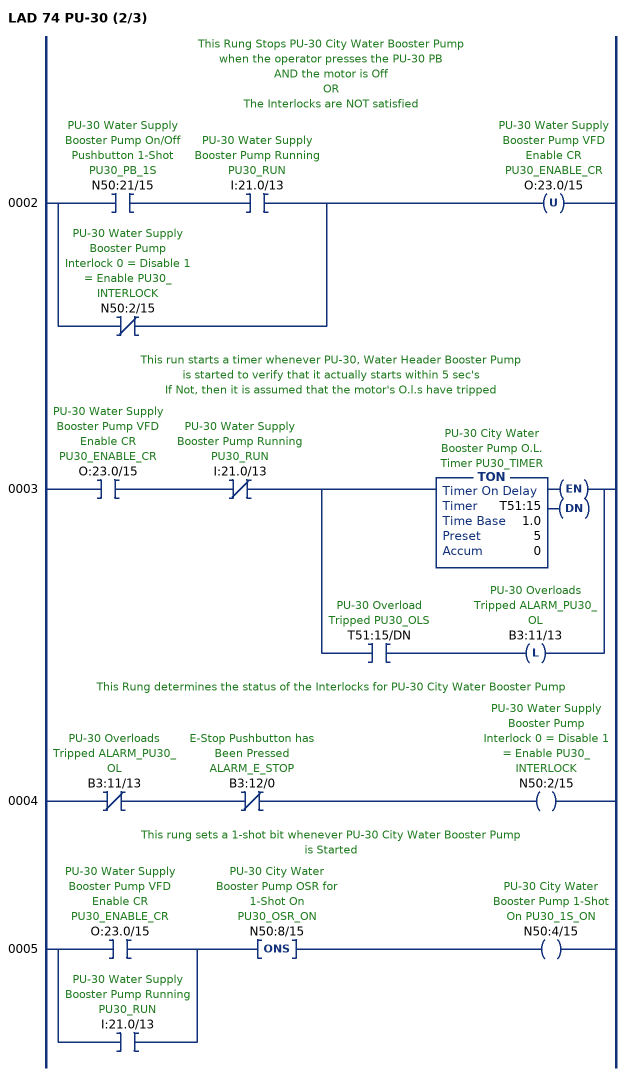
% Rung: 2 %
% This Rung Stops PU-30 City Water Booster Pump
% when the operator presses the PU-30 PB
% AND the motor is Off
% OR
% The Interlocks are NOT satisfied %
SOR BST XIC N50:21/15 XIC I:21.0/13 NXB XIO N50:2/15 BND OTU O:23.0/15 EOR
%   N50:21/15  PU30_PB_1S  "PU-30 Water Supply Booster Pump On/Off Pushbutton 1-Shot" %
%   I:21.0/13  PU30_RUN  "PU-30 Water Supply Booster Pump Running" %
%   N50:2/15  PU30_INTERLOCK  "PU-30 Water Supply Booster Pump Interlock 0 = Disable 1 = Enable" %
%   O:23.0/15  PU30_ENABLE_CR  "PU-30 Water Supply Booster Pump VFD Enable CR" %
% Rung: 3 %
% This run starts a timer whenever PU-30, Water Header Booster Pump
% is started to verify that it actually starts within 5 sec's
% If Not, then it is assumed that the motor's O.l.s have tripped %
SOR XIC O:23.0/15 XIO I:21.0/13 BST TON T51:15 1.0 5 0 NXB XIC T51:15/DN OTL B3:11/13 BND EOR
%   O:23.0/15  PU30_ENABLE_CR  "PU-30 Water Supply Booster Pump VFD Enable CR" %
%   I:21.0/13  PU30_RUN  "PU-30 Water Supply Booster Pump Running" %
%   T51:15  PU30_TIMER  "PU-30 City Water Booster Pump O.L. Timer" %
%   T51:15/DN  PU30_OLS  "PU-30 Overload Tripped" %
%   B3:11/13  ALARM_PU30_OL  "PU-30 Overloads Tripped" %
% Rung: 4 %
% This Rung determines the status of the Interlocks for PU-30 City Water Booster Pump %
SOR XIO B3:11/13 XIO B3:12/0 OTE N50:2/15 EOR
%   B3:11/13  ALARM_PU30_OL  "PU-30 Overloads Tripped" %
%   B3:12/0  ALARM_E_STOP  "E-Stop Pushbutton has Been Pressed" %
%   N50:2/15  PU30_INTERLOCK  "PU-30 Water Supply Booster Pump Interlock 0 = Disable 1 = Enable" %
% Rung: 5 %
% This rung sets a 1-shot bit whenever PU-30 City Water Booster Pump
% is Started %
SOR BST XIC O:23.0/15 NXB XIC I:21.0/13 BND OSR N50:8/15 OTE N50:4/15 EOR
%   O:23.0/15  PU30_ENABLE_CR  "PU-30 Water Supply Booster Pump VFD Enable CR" %
%   I:21.0/13  PU30_RUN  "PU-30 Water Supply Booster Pump Running" %
%   N50:8/15  PU30_OSR_ON  "PU-30 City Water Booster Pump OSR for 1-Shot On" %
%   N50:4/15  PU30_1S_ON  "PU-30 City Water Booster Pump 1-Shot On" %

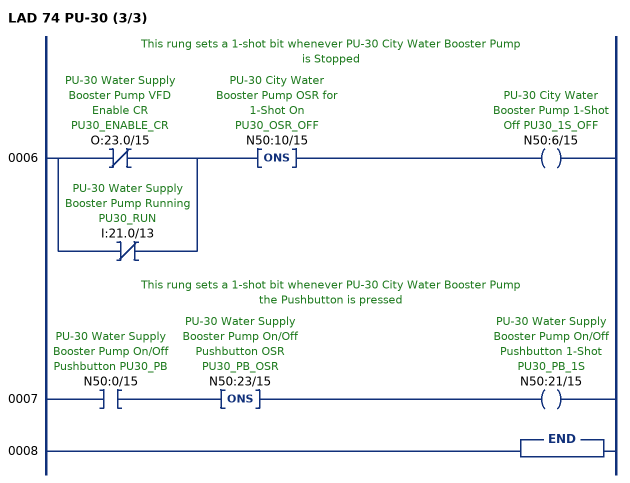
% Rung: 6 %
% This rung sets a 1-shot bit whenever PU-30 City Water Booster Pump
% is Stopped %
SOR BST XIO O:23.0/15 NXB XIO I:21.0/13 BND OSR N50:10/15 OTE N50:6/15 EOR
%   O:23.0/15  PU30_ENABLE_CR  "PU-30 Water Supply Booster Pump VFD Enable CR" %
%   I:21.0/13  PU30_RUN  "PU-30 Water Supply Booster Pump Running" %
%   N50:10/15  PU30_OSR_OFF  "PU-30 City Water Booster Pump OSR for 1-Shot On" %
%   N50:6/15  PU30_1S_OFF  "PU-30 City Water Booster Pump 1-Shot Off" %
% Rung: 7 %
% This rung sets a 1-shot bit whenever PU-30 City Water Booster Pump
% the Pushbutton is pressed %
SOR XIC N50:0/15 OSR N50:23/15 OTE N50:21/15 EOR
%   N50:0/15  PU30_PB  "PU-30 Water Supply Booster Pump On/Off Pushbutton" %
%   N50:23/15  PU30_PB_OSR  "PU-30 Water Supply Booster Pump On/Off Pushbutton OSR" %
%   N50:21/15  PU30_PB_1S  "PU-30 Water Supply Booster Pump On/Off Pushbutton 1-Shot" %
% Rung: 8 %
SOR END EOR

LADDER 75 "VB-35"    % VB-35 Tuthill Vacuum Blower Controls %
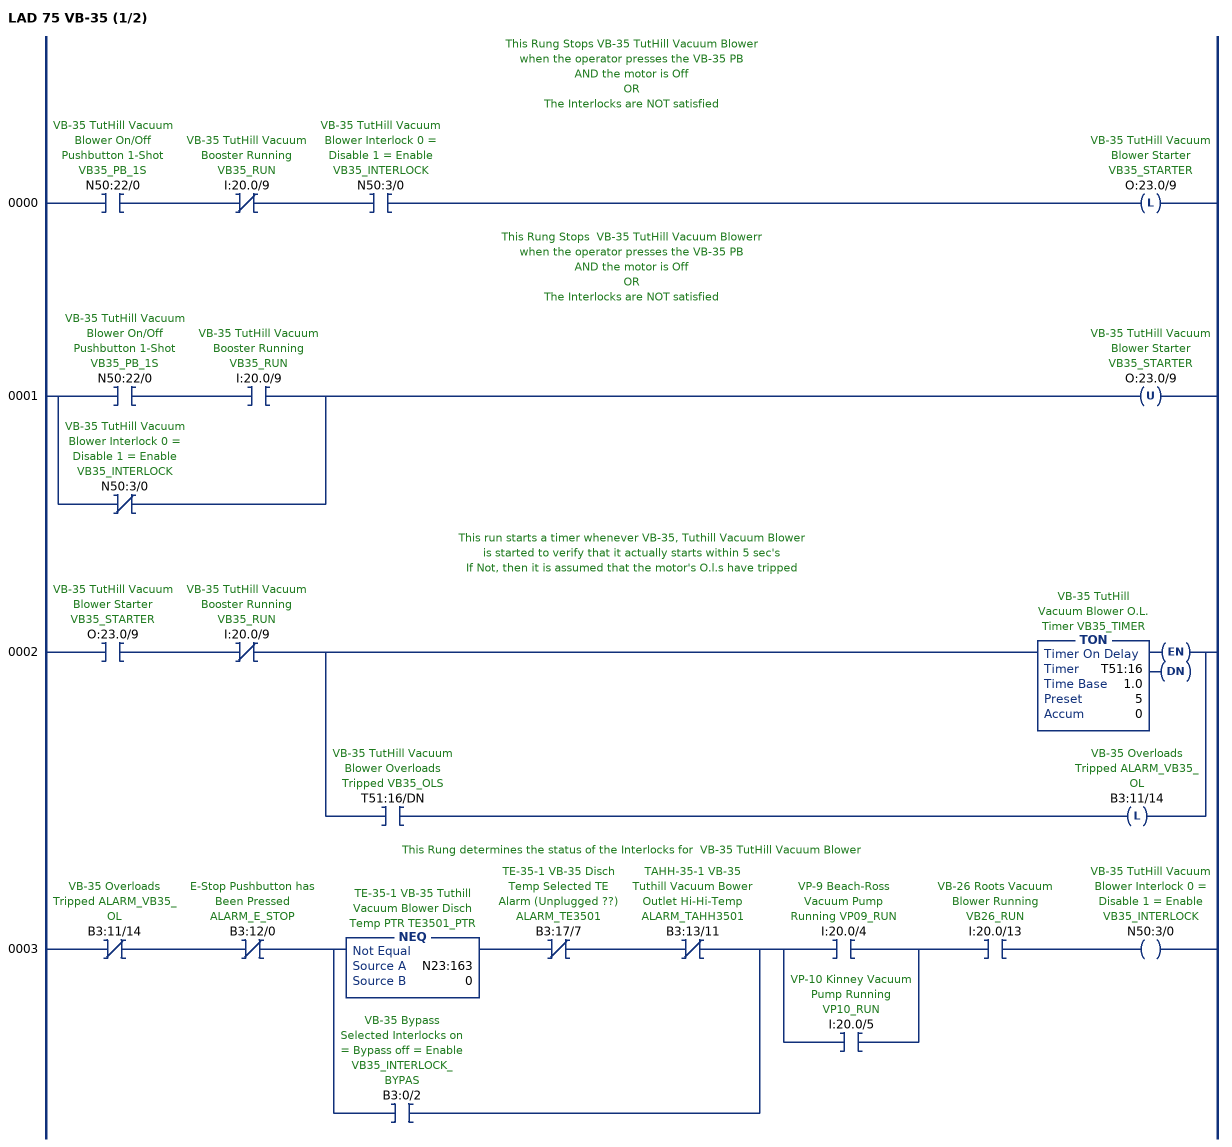
% Rung: 0 %
% This Rung Stops VB-35 TutHill Vacuum Blower
% when the operator presses the VB-35 PB
% AND the motor is Off
% OR
% The Interlocks are NOT satisfied %
SOR XIC N50:22/0 XIO I:20.0/9 XIC N50:3/0 OTL O:23.0/9 EOR
%   N50:22/0  VB35_PB_1S  "VB-35 TutHill Vacuum Blower On/Off Pushbutton 1-Shot" %
%   I:20.0/9  VB35_RUN  "VB-35 TutHill Vacuum Booster Running" %
%   N50:3/0  VB35_INTERLOCK  "VB-35 TutHill Vacuum Blower Interlock 0 = Disable 1 = Enable" %
%   O:23.0/9  VB35_STARTER  "VB-35 TutHill Vacuum Blower Starter" %
% Rung: 1 %
% This Rung Stops  VB-35 TutHill Vacuum Blowerr
% when the operator presses the VB-35 PB
% AND the motor is Off
% OR
% The Interlocks are NOT satisfied %
SOR BST XIC N50:22/0 XIC I:20.0/9 NXB XIO N50:3/0 BND OTU O:23.0/9 EOR
%   N50:22/0  VB35_PB_1S  "VB-35 TutHill Vacuum Blower On/Off Pushbutton 1-Shot" %
%   I:20.0/9  VB35_RUN  "VB-35 TutHill Vacuum Booster Running" %
%   N50:3/0  VB35_INTERLOCK  "VB-35 TutHill Vacuum Blower Interlock 0 = Disable 1 = Enable" %
%   O:23.0/9  VB35_STARTER  "VB-35 TutHill Vacuum Blower Starter" %
% Rung: 2 %
% This run starts a timer whenever VB-35, Tuthill Vacuum Blower
% is started to verify that it actually starts within 5 sec's
% If Not, then it is assumed that the motor's O.l.s have tripped %
SOR XIC O:23.0/9 XIO I:20.0/9 BST TON T51:16 1.0 5 0 NXB XIC T51:16/DN OTL B3:11/14 BND EOR
%   O:23.0/9  VB35_STARTER  "VB-35 TutHill Vacuum Blower Starter" %
%   I:20.0/9  VB35_RUN  "VB-35 TutHill Vacuum Booster Running" %
%   T51:16  VB35_TIMER  "VB-35 TutHill Vacuum Blower O.L. Timer" %
%   T51:16/DN  VB35_OLS  "VB-35 TutHill Vacuum Blower Overloads Tripped" %
%   B3:11/14  ALARM_VB35_OL  "VB-35 Overloads Tripped" %
% Rung: 3 %
% This Rung determines the status of the Interlocks for  VB-35 TutHill Vacuum Blower %
SOR XIO B3:11/14 XIO B3:12/0 BST NEQ N23:163 0 XIO B3:17/7 XIO B3:13/11 NXB XIC B3:0/2 BND BST XIC I:20.0/4 NXB XIC I:20.0/5 BND XIC I:20.0/13 OTE N50:3/0 EOR
%   B3:11/14  ALARM_VB35_OL  "VB-35 Overloads Tripped" %
%   B3:12/0  ALARM_E_STOP  "E-Stop Pushbutton has Been Pressed" %
%   N23:163  TE3501_PTR  "TE-35-1 VB-35 Tuthill Vacuum Blower Disch Temp PTR" %
%   B3:17/7  ALARM_TE3501  "TE-35-1 VB-35 Disch Temp Selected TE Alarm (Unplugged ??)" %
%   B3:13/11  ALARM_TAHH3501  "TAHH-35-1 VB-35 Tuthill Vacuum Bower Outlet Hi-Hi-Temp" %
%   B3:0/2  VB35_INTERLOCK_BYPAS  "VB-35 Bypass Selected Interlocks on = Bypass off = Enable" %
%   I:20.0/4  VP09_RUN  "VP-9 Beach-Ross Vacuum Pump Running" %
%   I:20.0/5  VP10_RUN  "VP-10 Kinney Vacuum Pump Running" %
%   I:20.0/13  VB26_RUN  "VB-26 Roots Vacuum Blower Running" %
%   N50:3/0  VB35_INTERLOCK  "VB-35 TutHill Vacuum Blower Interlock 0 = Disable 1 = Enable" %

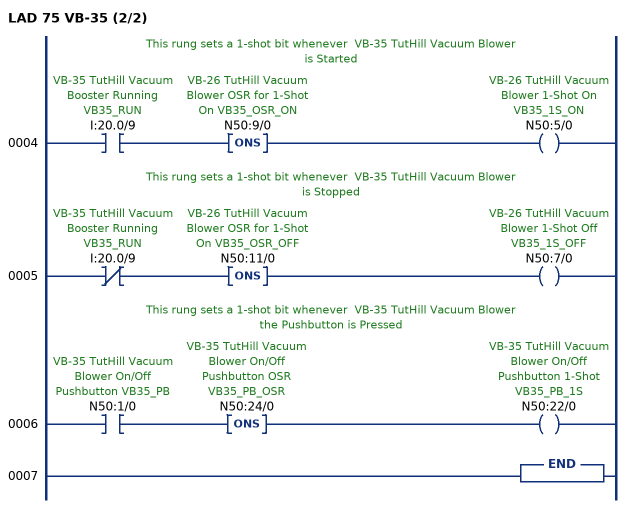
% Rung: 4 %
% This rung sets a 1-shot bit whenever  VB-35 TutHill Vacuum Blower
% is Started %
SOR XIC I:20.0/9 OSR N50:9/0 OTE N50:5/0 EOR
%   I:20.0/9  VB35_RUN  "VB-35 TutHill Vacuum Booster Running" %
%   N50:9/0  VB35_OSR_ON  "VB-26 TutHill Vacuum Blower OSR for 1-Shot On" %
%   N50:5/0  VB35_1S_ON  "VB-26 TutHill Vacuum Blower 1-Shot On" %
% Rung: 5 %
% This rung sets a 1-shot bit whenever  VB-35 TutHill Vacuum Blower
% is Stopped %
SOR XIO I:20.0/9 OSR N50:11/0 OTE N50:7/0 EOR
%   I:20.0/9  VB35_RUN  "VB-35 TutHill Vacuum Booster Running" %
%   N50:11/0  VB35_OSR_OFF  "VB-26 TutHill Vacuum Blower OSR for 1-Shot On" %
%   N50:7/0  VB35_1S_OFF  "VB-26 TutHill Vacuum Blower 1-Shot Off" %
% Rung: 6 %
% This rung sets a 1-shot bit whenever  VB-35 TutHill Vacuum Blower
% the Pushbutton is Pressed %
SOR XIC N50:1/0 OSR N50:24/0 OTE N50:22/0 EOR
%   N50:1/0  VB35_PB  "VB-35 TutHill Vacuum Blower On/Off Pushbutton" %
%   N50:24/0  VB35_PB_OSR  "VB-35 TutHill Vacuum Blower On/Off Pushbutton OSR" %
%   N50:22/0  VB35_PB_1S  "VB-35 TutHill Vacuum Blower On/Off Pushbutton 1-Shot" %
% Rung: 7 %
SOR END EOR

LADDER 77 "PU-37"    % PU-37, Temperaed Oil No-3 Controls %
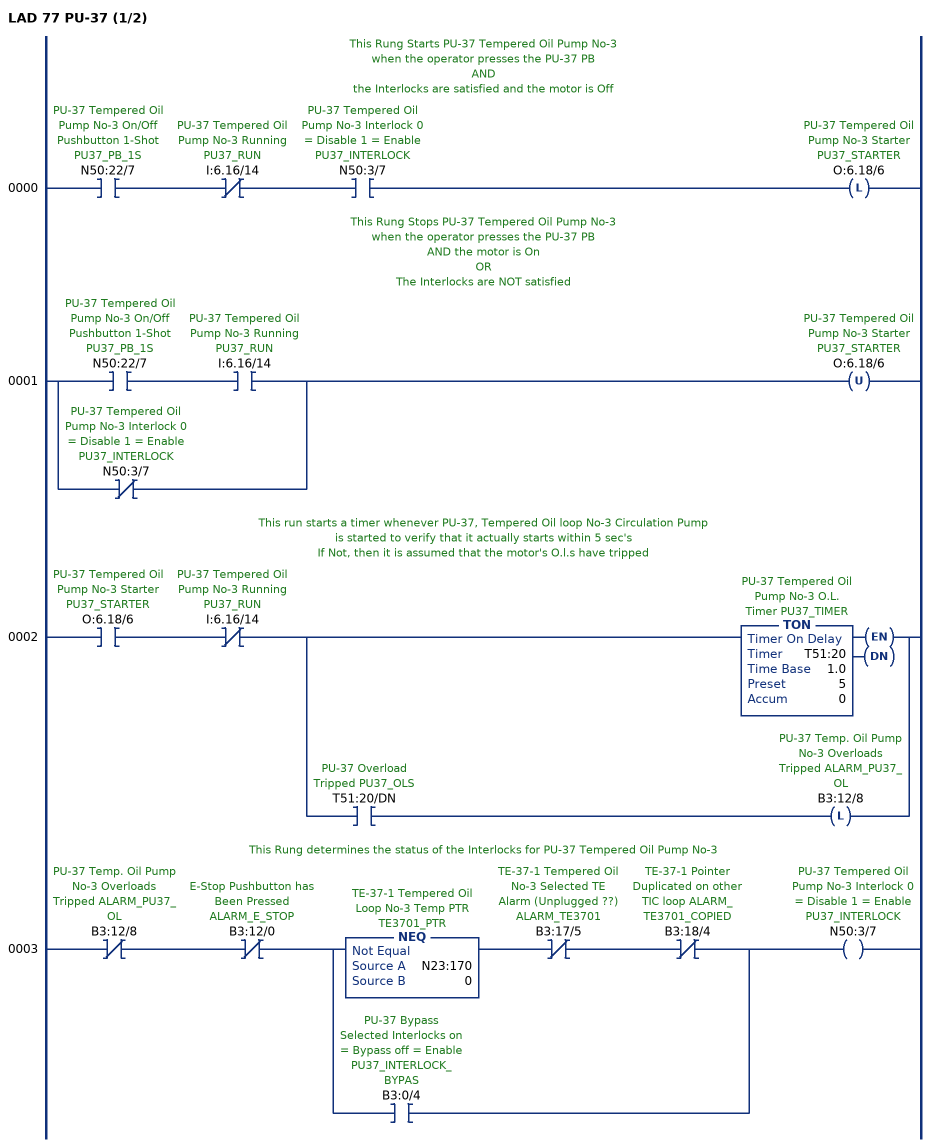
% Rung: 0 %
% This Rung Starts PU-37 Tempered Oil Pump No-3
% when the operator presses the PU-37 PB
% AND
% the Interlocks are satisfied and the motor is Off %
SOR XIC N50:22/7 XIO I:6.16/14 XIC N50:3/7 OTL O:6.18/6 EOR
%   N50:22/7  PU37_PB_1S  "PU-37 Tempered Oil Pump No-3 On/Off Pushbutton 1-Shot" %
%   I:6.16/14  PU37_RUN  "PU-37 Tempered Oil Pump No-3 Running" %
%   N50:3/7  PU37_INTERLOCK  "PU-37 Tempered Oil Pump No-3 Interlock 0 = Disable 1 = Enable" %
%   O:6.18/6  PU37_STARTER  "PU-37 Tempered Oil Pump No-3 Starter" %
% Rung: 1 %
% This Rung Stops PU-37 Tempered Oil Pump No-3
% when the operator presses the PU-37 PB
% AND the motor is On
% OR
% The Interlocks are NOT satisfied %
SOR BST XIC N50:22/7 XIC I:6.16/14 NXB XIO N50:3/7 BND OTU O:6.18/6 EOR
%   N50:22/7  PU37_PB_1S  "PU-37 Tempered Oil Pump No-3 On/Off Pushbutton 1-Shot" %
%   I:6.16/14  PU37_RUN  "PU-37 Tempered Oil Pump No-3 Running" %
%   N50:3/7  PU37_INTERLOCK  "PU-37 Tempered Oil Pump No-3 Interlock 0 = Disable 1 = Enable" %
%   O:6.18/6  PU37_STARTER  "PU-37 Tempered Oil Pump No-3 Starter" %
% Rung: 2 %
% This run starts a timer whenever PU-37, Tempered Oil loop No-3 Circulation Pump
% is started to verify that it actually starts within 5 sec's
% If Not, then it is assumed that the motor's O.l.s have tripped %
SOR XIC O:6.18/6 XIO I:6.16/14 BST TON T51:20 1.0 5 0 NXB XIC T51:20/DN OTL B3:12/8 BND EOR
%   O:6.18/6  PU37_STARTER  "PU-37 Tempered Oil Pump No-3 Starter" %
%   I:6.16/14  PU37_RUN  "PU-37 Tempered Oil Pump No-3 Running" %
%   T51:20  PU37_TIMER  "PU-37 Tempered Oil Pump No-3 O.L. Timer" %
%   T51:20/DN  PU37_OLS  "PU-37 Overload Tripped" %
%   B3:12/8  ALARM_PU37_OL  "PU-37 Temp. Oil Pump No-3 Overloads Tripped" %
% Rung: 3 %
% This Rung determines the status of the Interlocks for PU-37 Tempered Oil Pump No-3 %
SOR XIO B3:12/8 XIO B3:12/0 BST NEQ N23:170 0 XIO B3:17/5 XIO B3:18/4 NXB XIC B3:0/4 BND OTE N50:3/7 EOR
%   B3:12/8  ALARM_PU37_OL  "PU-37 Temp. Oil Pump No-3 Overloads Tripped" %
%   B3:12/0  ALARM_E_STOP  "E-Stop Pushbutton has Been Pressed" %
%   N23:170  TE3701_PTR  "TE-37-1 Tempered Oil Loop No-3 Temp PTR" %
%   B3:17/5  ALARM_TE3701  "TE-37-1 Tempered Oil No-3 Selected TE Alarm (Unplugged ??)" %
%   B3:18/4  ALARM_TE3701_COPIED  "TE-37-1 Pointer Duplicated on other TIC loop" %
%   B3:0/4  PU37_INTERLOCK_BYPAS  "PU-37 Bypass Selected Interlocks on = Bypass off = Enable" %
%   N50:3/7  PU37_INTERLOCK  "PU-37 Tempered Oil Pump No-3 Interlock 0 = Disable 1 = Enable" %

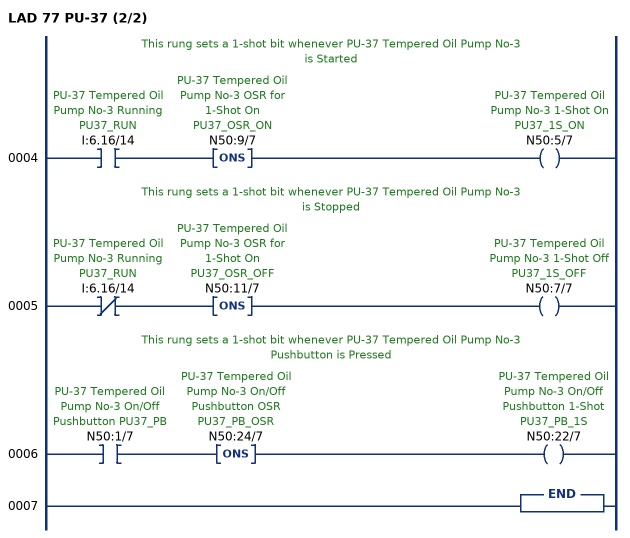
% Rung: 4 %
% This rung sets a 1-shot bit whenever PU-37 Tempered Oil Pump No-3
% is Started %
SOR XIC I:6.16/14 OSR N50:9/7 OTE N50:5/7 EOR
%   I:6.16/14  PU37_RUN  "PU-37 Tempered Oil Pump No-3 Running" %
%   N50:9/7  PU37_OSR_ON  "PU-37 Tempered Oil Pump No-3 OSR for 1-Shot On" %
%   N50:5/7  PU37_1S_ON  "PU-37 Tempered Oil Pump No-3 1-Shot On" %
% Rung: 5 %
% This rung sets a 1-shot bit whenever PU-37 Tempered Oil Pump No-3
% is Stopped %
SOR XIO I:6.16/14 OSR N50:11/7 OTE N50:7/7 EOR
%   I:6.16/14  PU37_RUN  "PU-37 Tempered Oil Pump No-3 Running" %
%   N50:11/7  PU37_OSR_OFF  "PU-37 Tempered Oil Pump No-3 OSR for 1-Shot On" %
%   N50:7/7  PU37_1S_OFF  "PU-37 Tempered Oil Pump No-3 1-Shot Off" %
% Rung: 6 %
% This rung sets a 1-shot bit whenever PU-37 Tempered Oil Pump No-3
% Pushbutton is Pressed %
SOR XIC N50:1/7 OSR N50:24/7 OTE N50:22/7 EOR
%   N50:1/7  PU37_PB  "PU-37 Tempered Oil Pump No-3 On/Off Pushbutton" %
%   N50:24/7  PU37_PB_OSR  "PU-37 Tempered Oil Pump No-3 On/Off Pushbutton OSR" %
%   N50:22/7  PU37_PB_1S  "PU-37 Tempered Oil Pump No-3 On/Off Pushbutton 1-Shot" %
% Rung: 7 %
SOR END EOR

LADDER 80 "PU-40"    % PU-40, Temperaed Oil No-2 Controls %
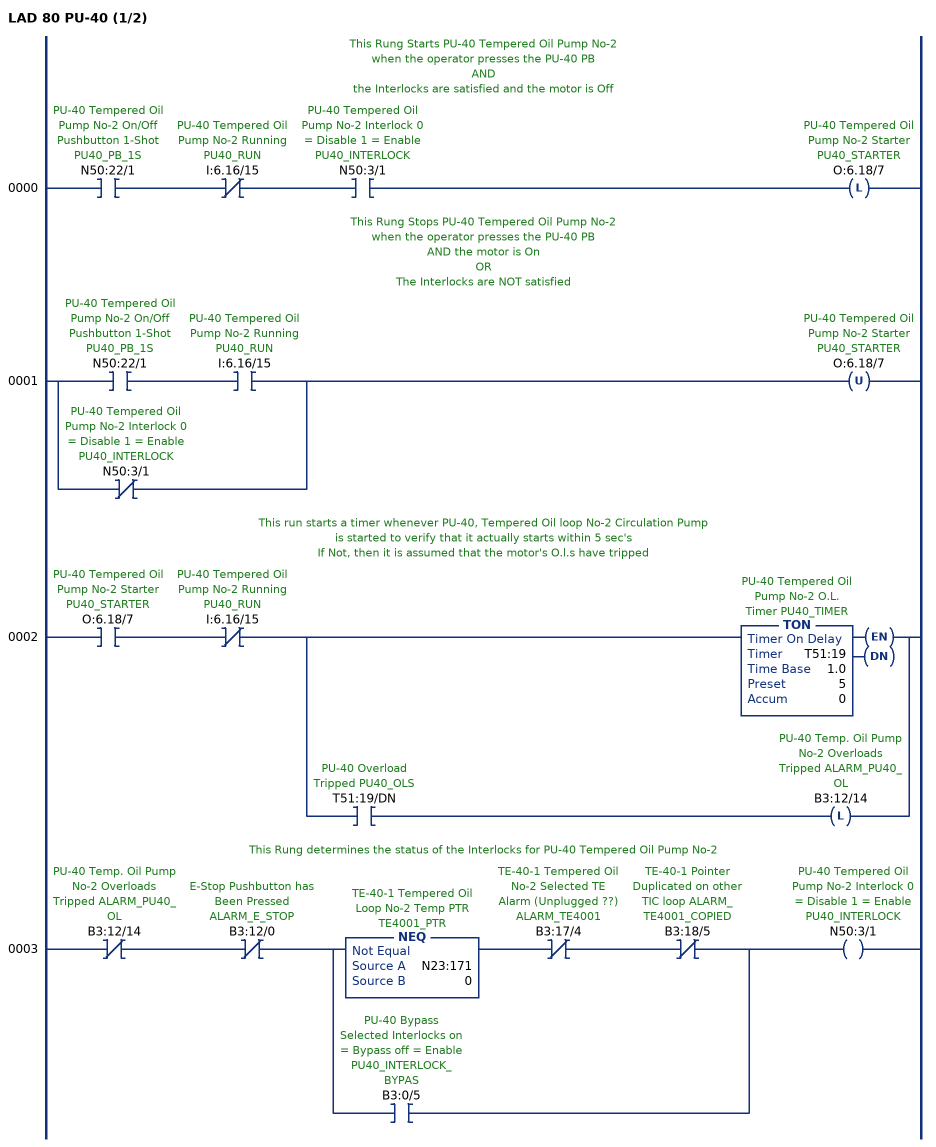
% Rung: 0 %
% This Rung Starts PU-40 Tempered Oil Pump No-2
% when the operator presses the PU-40 PB
% AND
% the Interlocks are satisfied and the motor is Off %
SOR XIC N50:22/1 XIO I:6.16/15 XIC N50:3/1 OTL O:6.18/7 EOR
%   N50:22/1  PU40_PB_1S  "PU-40 Tempered Oil Pump No-2 On/Off Pushbutton 1-Shot" %
%   I:6.16/15  PU40_RUN  "PU-40 Tempered Oil Pump No-2 Running" %
%   N50:3/1  PU40_INTERLOCK  "PU-40 Tempered Oil Pump No-2 Interlock 0 = Disable 1 = Enable" %
%   O:6.18/7  PU40_STARTER  "PU-40 Tempered Oil Pump No-2 Starter" %
% Rung: 1 %
% This Rung Stops PU-40 Tempered Oil Pump No-2
% when the operator presses the PU-40 PB
% AND the motor is On
% OR
% The Interlocks are NOT satisfied %
SOR BST XIC N50:22/1 XIC I:6.16/15 NXB XIO N50:3/1 BND OTU O:6.18/7 EOR
%   N50:22/1  PU40_PB_1S  "PU-40 Tempered Oil Pump No-2 On/Off Pushbutton 1-Shot" %
%   I:6.16/15  PU40_RUN  "PU-40 Tempered Oil Pump No-2 Running" %
%   N50:3/1  PU40_INTERLOCK  "PU-40 Tempered Oil Pump No-2 Interlock 0 = Disable 1 = Enable" %
%   O:6.18/7  PU40_STARTER  "PU-40 Tempered Oil Pump No-2 Starter" %
% Rung: 2 %
% This run starts a timer whenever PU-40, Tempered Oil loop No-2 Circulation Pump
% is started to verify that it actually starts within 5 sec's
% If Not, then it is assumed that the motor's O.l.s have tripped %
SOR XIC O:6.18/7 XIO I:6.16/15 BST TON T51:19 1.0 5 0 NXB XIC T51:19/DN OTL B3:12/14 BND EOR
%   O:6.18/7  PU40_STARTER  "PU-40 Tempered Oil Pump No-2 Starter" %
%   I:6.16/15  PU40_RUN  "PU-40 Tempered Oil Pump No-2 Running" %
%   T51:19  PU40_TIMER  "PU-40 Tempered Oil Pump No-2 O.L. Timer" %
%   T51:19/DN  PU40_OLS  "PU-40 Overload Tripped" %
%   B3:12/14  ALARM_PU40_OL  "PU-40 Temp. Oil Pump No-2 Overloads Tripped" %
% Rung: 3 %
% This Rung determines the status of the Interlocks for PU-40 Tempered Oil Pump No-2 %
SOR XIO B3:12/14 XIO B3:12/0 BST NEQ N23:171 0 XIO B3:17/4 XIO B3:18/5 NXB XIC B3:0/5 BND OTE N50:3/1 EOR
%   B3:12/14  ALARM_PU40_OL  "PU-40 Temp. Oil Pump No-2 Overloads Tripped" %
%   B3:12/0  ALARM_E_STOP  "E-Stop Pushbutton has Been Pressed" %
%   N23:171  TE4001_PTR  "TE-40-1 Tempered Oil Loop No-2 Temp PTR" %
%   B3:17/4  ALARM_TE4001  "TE-40-1 Tempered Oil No-2 Selected TE Alarm (Unplugged ??)" %
%   B3:18/5  ALARM_TE4001_COPIED  "TE-40-1 Pointer Duplicated on other TIC loop" %
%   B3:0/5  PU40_INTERLOCK_BYPAS  "PU-40 Bypass Selected Interlocks on = Bypass off = Enable" %
%   N50:3/1  PU40_INTERLOCK  "PU-40 Tempered Oil Pump No-2 Interlock 0 = Disable 1 = Enable" %

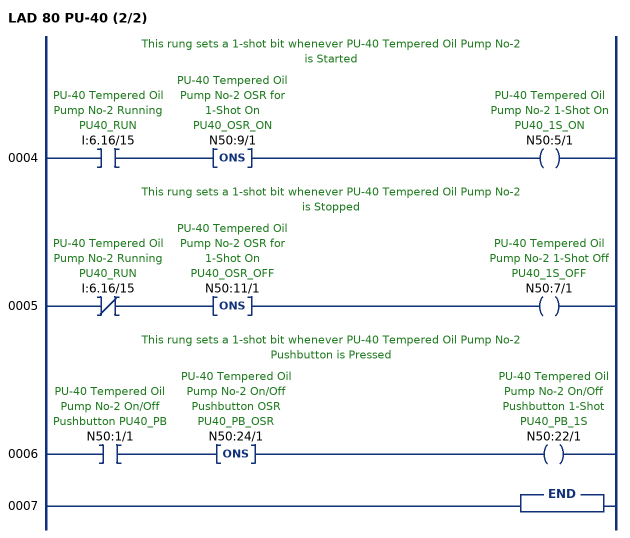
% Rung: 4 %
% This rung sets a 1-shot bit whenever PU-40 Tempered Oil Pump No-2
% is Started %
SOR XIC I:6.16/15 OSR N50:9/1 OTE N50:5/1 EOR
%   I:6.16/15  PU40_RUN  "PU-40 Tempered Oil Pump No-2 Running" %
%   N50:9/1  PU40_OSR_ON  "PU-40 Tempered Oil Pump No-2 OSR for 1-Shot On" %
%   N50:5/1  PU40_1S_ON  "PU-40 Tempered Oil Pump No-2 1-Shot On" %
% Rung: 5 %
% This rung sets a 1-shot bit whenever PU-40 Tempered Oil Pump No-2
% is Stopped %
SOR XIO I:6.16/15 OSR N50:11/1 OTE N50:7/1 EOR
%   I:6.16/15  PU40_RUN  "PU-40 Tempered Oil Pump No-2 Running" %
%   N50:11/1  PU40_OSR_OFF  "PU-40 Tempered Oil Pump No-2 OSR for 1-Shot On" %
%   N50:7/1  PU40_1S_OFF  "PU-40 Tempered Oil Pump No-2 1-Shot Off" %
% Rung: 6 %
% This rung sets a 1-shot bit whenever PU-40 Tempered Oil Pump No-2
% Pushbutton is Pressed %
SOR XIC N50:1/1 OSR N50:24/1 OTE N50:22/1 EOR
%   N50:1/1  PU40_PB  "PU-40 Tempered Oil Pump No-2 On/Off Pushbutton" %
%   N50:24/1  PU40_PB_OSR  "PU-40 Tempered Oil Pump No-2 On/Off Pushbutton OSR" %
%   N50:22/1  PU40_PB_1S  "PU-40 Tempered Oil Pump No-2 On/Off Pushbutton 1-Shot" %
% Rung: 7 %
SOR END EOR

LADDER 81 "EV-42"    % EV-42 Rotor Drive VFD Controls %
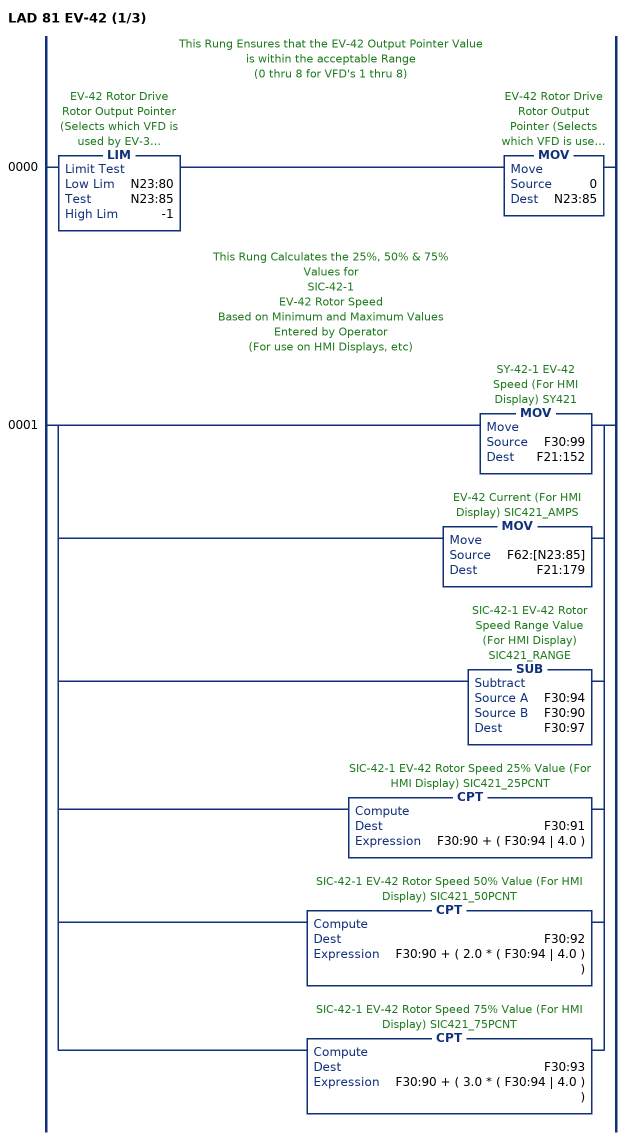
% Rung: 0 %
% This Rung Ensures that the EV-42 Output Pointer Value
% is within the acceptable Range
% (0 thru 8 for VFD's 1 thru 8) %
SOR LIM N23:80 N23:85 -1 MOV 0 N23:85 EOR
%   N23:80  MAX_VFD_ALLOWED_1  "Maximum Number of VFDs Available Plus 1" %
%   N23:85  EV42_OUT_PTR  "EV-42 Rotor Drive Rotor Output Pointer (Selects which VFD is used by EV-3)" %
% Rung: 1 %
% This Rung Calculates the 25%, 50% & 75%
% Values for
% SIC-42-1
% EV-42 Rotor Speed
% Based on Minimum and Maximum Values
% Entered by Operator
% (For use on HMI Displays, etc) %
SOR BST MOV F30:99 F21:152 NXB MOV F62:[N23:85] F21:179 NXB SUB F30:94 F30:90 F30:97 NXB CPT F30:91 " F30:90 + ( F30:94 | 4.0 ) " NXB CPT F30:92 " F30:90 + ( 2.0 * ( F30:94 | 4.0 ) ) " NXB CPT F30:93 " F30:90 + ( 3.0 * ( F30:94 | 4.0 ) ) " BND EOR
%   F30:99  SIC421_SP_FP  "SIC-42-1 EV-42 Rotor Speed Setpoint Value (For HMI Display)" %
%   F21:152  SY421  "SY-42-1 EV-42 Speed (For HMI Display)" %
%   N23:85  EV42_OUT_PTR  "EV-42 Rotor Drive Rotor Output Pointer (Selects which VFD is used by EV-3)" %
%   F21:179  SIC421_AMPS  "EV-42 Current (For HMI Display)" %
%   F30:94  SIC421_MAX  "SIC-42-1 EV-42 Rotor Speed 100% Value (For HMI Display)" %
%   F30:90  SIC421_MIN  "SIC-42-1 EV-42 Rotor Speed 0% Value (For HMI Display)" %
%   F30:97  SIC421_RANGE  "SIC-42-1 EV-42 Rotor Speed Range Value (For HMI Display)" %
%   F30:91  SIC421_25PCNT  "SIC-42-1 EV-42 Rotor Speed 25% Value (For HMI Display)" %
%   F30:92  SIC421_50PCNT  "SIC-42-1 EV-42 Rotor Speed 50% Value (For HMI Display)" %
%   F30:93  SIC421_75PCNT  "SIC-42-1 EV-42 Rotor Speed 75% Value (For HMI Display)" %

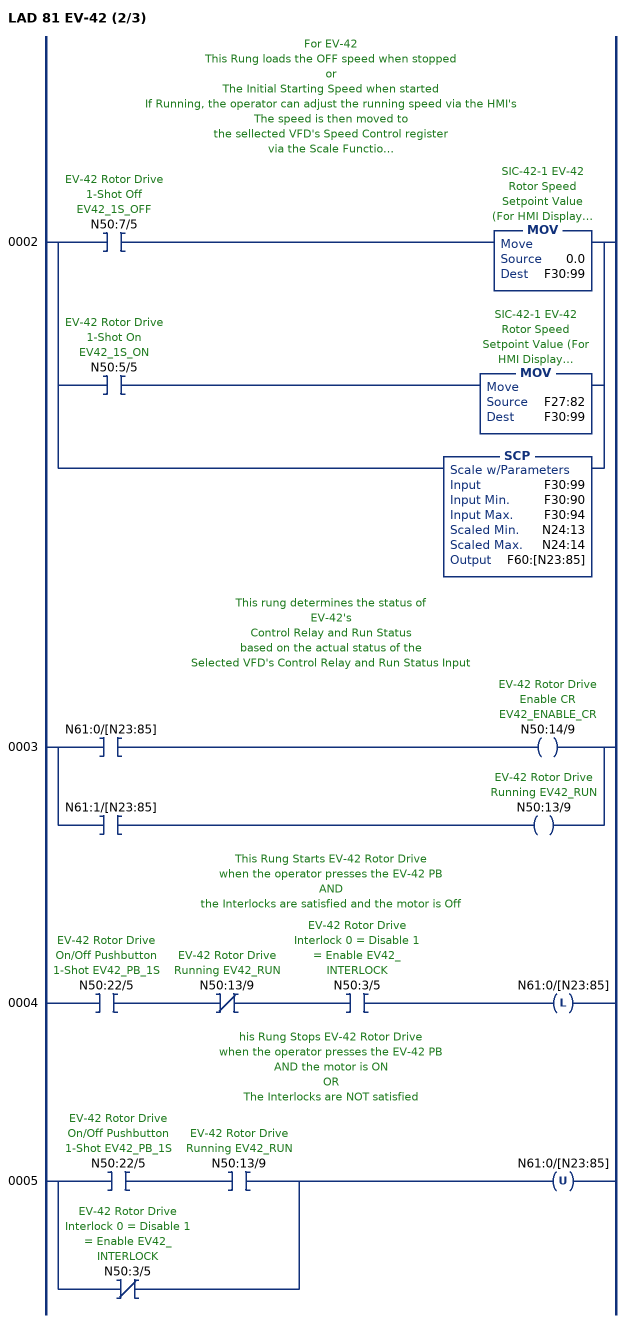
% Rung: 2 %
% For EV-42
% This Rung loads the OFF speed when stopped
% or
% The Initial Starting Speed when started
% If Running, the operator can adjust the running speed via the HMI's
% The speed is then moved to
% the sellected VFD's Speed Control register
% via the Scale Function
% to actually adjust the VFD's Speed %
SOR BST XIC N50:7/5 MOV 0.0 F30:99 NXB XIC N50:5/5 MOV F27:82 F30:99 NXB SCP F30:99 F30:90 F30:94 N24:13 N24:14 F60:[N23:85] BND EOR
%   N50:7/5  EV42_1S_OFF  "EV-42 Rotor Drive 1-Shot Off" %
%   F30:99  SIC421_SP_FP  "SIC-42-1 EV-42 Rotor Speed Setpoint Value (For HMI Display)" %
%   N50:5/5  EV42_1S_ON  "EV-42 Rotor Drive 1-Shot On" %
%   F27:82  SIC421_INIT_SP  "SY-42-1 Initial Speed Setpoint (RPM)" %
%   F30:90  SIC421_MIN  "SIC-42-1 EV-42 Rotor Speed 0% Value (For HMI Display)" %
%   F30:94  SIC421_MAX  "SIC-42-1 EV-42 Rotor Speed 100% Value (For HMI Display)" %
%   N24:13  AO_MIN_OE4  "Analog Output Minimum Value Generates 4 mA DC (To OE4 AO Module)" %
%   N24:14  AO_MAX_OE4  "Analog Output Maximum Value Generates 20 mA DC (To OE4 AO Module)" %
%   N23:85  EV42_OUT_PTR  "EV-42 Rotor Drive Rotor Output Pointer (Selects which VFD is used by EV-3)" %
% Rung: 3 %
% This rung determines the status of
% EV-42's
% Control Relay and Run Status
% based on the actual status of the
% Selected VFD's Control Relay and Run Status Input %
SOR BST XIC N61:0/[N23:85] OTE N50:14/9 NXB XIC N61:1/[N23:85] OTE N50:13/9 BND EOR
%   N61:0  VFD_ENABLE_BITS  "These Bits Enable the appropriate VFD" %
%   N23:85  EV42_OUT_PTR  "EV-42 Rotor Drive Rotor Output Pointer (Selects which VFD is used by EV-3)" %
%   N50:14/9  EV42_ENABLE_CR  "EV-42 Rotor Drive Enable CR" %
%   N61:1  VFD_RUN_BITS_1  "These Bits Initcate the Status Off/Running for the appropriate VFD" %
%   N50:13/9  EV42_RUN  "EV-42 Rotor Drive Running" %
% Rung: 4 %
% This Rung Starts EV-42 Rotor Drive
% when the operator presses the EV-42 PB
% AND
% the Interlocks are satisfied and the motor is Off %
SOR XIC N50:22/5 XIO N50:13/9 XIC N50:3/5 OTL N61:0/[N23:85] EOR
%   N50:22/5  EV42_PB_1S  "EV-42 Rotor Drive On/Off Pushbutton 1-Shot" %
%   N50:13/9  EV42_RUN  "EV-42 Rotor Drive Running" %
%   N50:3/5  EV42_INTERLOCK  "EV-42 Rotor Drive Interlock 0 = Disable 1 = Enable" %
%   N61:0  VFD_ENABLE_BITS  "These Bits Enable the appropriate VFD" %
%   N23:85  EV42_OUT_PTR  "EV-42 Rotor Drive Rotor Output Pointer (Selects which VFD is used by EV-3)" %
% Rung: 5 %
% his Rung Stops EV-42 Rotor Drive
% when the operator presses the EV-42 PB
% AND the motor is ON
% OR
% The Interlocks are NOT satisfied %
SOR BST XIC N50:22/5 XIC N50:13/9 NXB XIO N50:3/5 BND OTU N61:0/[N23:85] EOR
%   N50:22/5  EV42_PB_1S  "EV-42 Rotor Drive On/Off Pushbutton 1-Shot" %
%   N50:13/9  EV42_RUN  "EV-42 Rotor Drive Running" %
%   N50:3/5  EV42_INTERLOCK  "EV-42 Rotor Drive Interlock 0 = Disable 1 = Enable" %
%   N61:0  VFD_ENABLE_BITS  "These Bits Enable the appropriate VFD" %
%   N23:85  EV42_OUT_PTR  "EV-42 Rotor Drive Rotor Output Pointer (Selects which VFD is used by EV-3)" %

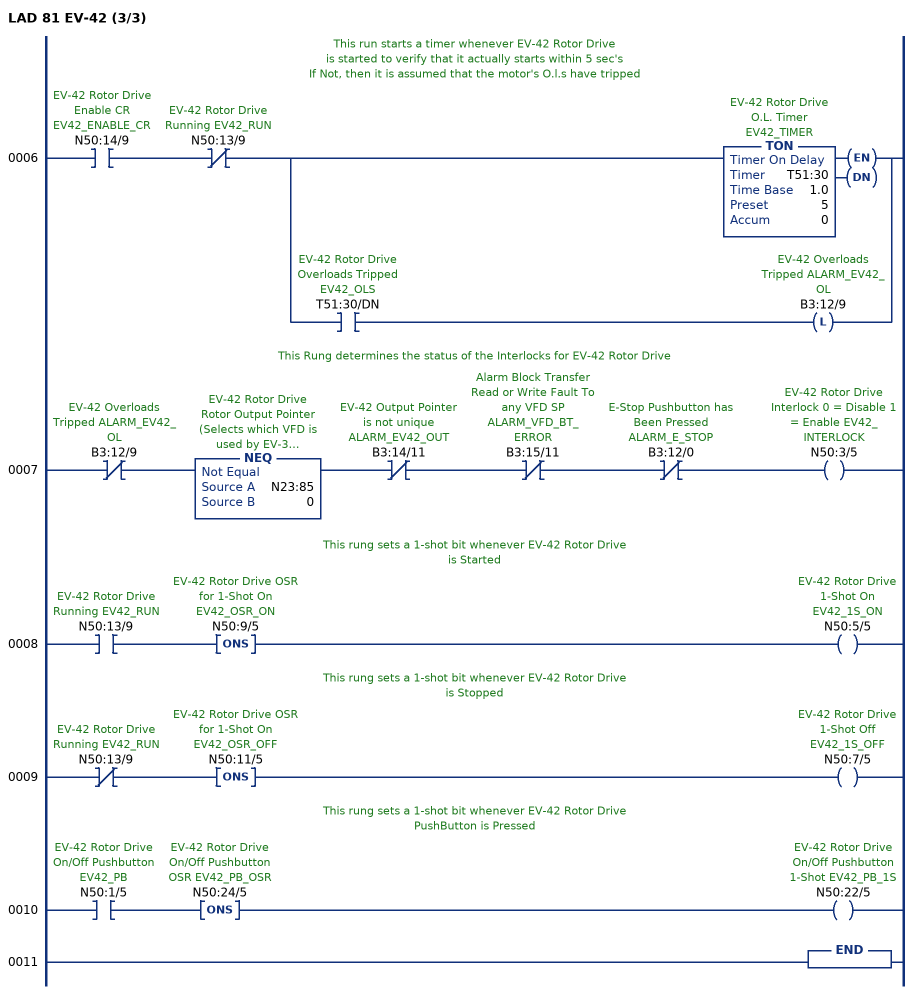
% Rung: 6 %
% This run starts a timer whenever EV-42 Rotor Drive
% is started to verify that it actually starts within 5 sec's
% If Not, then it is assumed that the motor's O.l.s have tripped %
SOR XIC N50:14/9 XIO N50:13/9 BST TON T51:30 1.0 5 0 NXB XIC T51:30/DN OTL B3:12/9 BND EOR
%   N50:14/9  EV42_ENABLE_CR  "EV-42 Rotor Drive Enable CR" %
%   N50:13/9  EV42_RUN  "EV-42 Rotor Drive Running" %
%   T51:30  EV42_TIMER  "EV-42 Rotor Drive O.L. Timer" %
%   T51:30/DN  EV42_OLS  "EV-42 Rotor Drive Overloads Tripped" %
%   B3:12/9  ALARM_EV42_OL  "EV-42 Overloads Tripped" %
% Rung: 7 %
% This Rung determines the status of the Interlocks for EV-42 Rotor Drive %
SOR XIO B3:12/9 NEQ N23:85 0 XIO B3:14/11 XIO B3:15/11 XIO B3:12/0 OTE N50:3/5 EOR
%   B3:12/9  ALARM_EV42_OL  "EV-42 Overloads Tripped" %
%   N23:85  EV42_OUT_PTR  "EV-42 Rotor Drive Rotor Output Pointer (Selects which VFD is used by EV-3)" %
%   B3:14/11  ALARM_EV42_OUT  "EV-42 Output Pointer is not unique" %
%   B3:15/11  ALARM_VFD_BT_ERROR  "Alarm Block Transfer Read or Write Fault To any VFD SP" %
%   B3:12/0  ALARM_E_STOP  "E-Stop Pushbutton has Been Pressed" %
%   N50:3/5  EV42_INTERLOCK  "EV-42 Rotor Drive Interlock 0 = Disable 1 = Enable" %
% Rung: 8 %
% This rung sets a 1-shot bit whenever EV-42 Rotor Drive
% is Started %
SOR XIC N50:13/9 OSR N50:9/5 OTE N50:5/5 EOR
%   N50:13/9  EV42_RUN  "EV-42 Rotor Drive Running" %
%   N50:9/5  EV42_OSR_ON  "EV-42 Rotor Drive OSR for 1-Shot On" %
%   N50:5/5  EV42_1S_ON  "EV-42 Rotor Drive 1-Shot On" %
% Rung: 9 %
% This rung sets a 1-shot bit whenever EV-42 Rotor Drive
% is Stopped %
SOR XIO N50:13/9 OSR N50:11/5 OTE N50:7/5 EOR
%   N50:13/9  EV42_RUN  "EV-42 Rotor Drive Running" %
%   N50:11/5  EV42_OSR_OFF  "EV-42 Rotor Drive OSR for 1-Shot On" %
%   N50:7/5  EV42_1S_OFF  "EV-42 Rotor Drive 1-Shot Off" %
% Rung: 10 %
% This rung sets a 1-shot bit whenever EV-42 Rotor Drive
% PushButton is Pressed %
SOR XIC N50:1/5 OSR N50:24/5 OTE N50:22/5 EOR
%   N50:1/5  EV42_PB  "EV-42 Rotor Drive On/Off Pushbutton" %
%   N50:24/5  EV42_PB_OSR  "EV-42 Rotor Drive On/Off Pushbutton OSR" %
%   N50:22/5  EV42_PB_1S  "EV-42 Rotor Drive On/Off Pushbutton 1-Shot" %
% Rung: 11 %
SOR END EOR

LADDER 82 "PU-46"    % PU-46, Flash Evaporator Circ Pump %
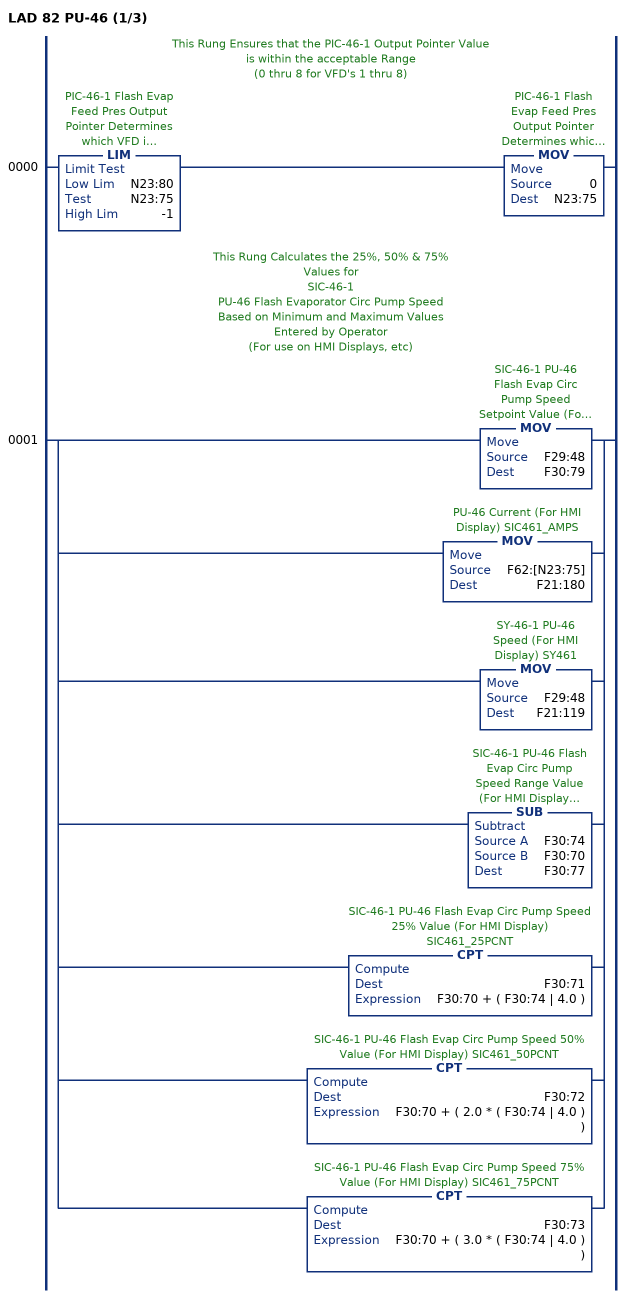
% Rung: 0 %
% This Rung Ensures that the PIC-46-1 Output Pointer Value
% is within the acceptable Range
% (0 thru 8 for VFD's 1 thru 8) %
SOR LIM N23:80 N23:75 -1 MOV 0 N23:75 EOR
%   N23:80  MAX_VFD_ALLOWED_1  "Maximum Number of VFDs Available Plus 1" %
%   N23:75  PIC461_OUT_PTR  "PIC-46-1 Flash Evap Feed Pres Output Pointer Determines which VFD is controled by FIC" %
% Rung: 1 %
% This Rung Calculates the 25%, 50% & 75%
% Values for
% SIC-46-1
% PU-46 Flash Evaporator Circ Pump Speed
% Based on Minimum and Maximum Values
% Entered by Operator
% (For use on HMI Displays, etc) %
SOR BST MOV F29:48 F30:79 NXB MOV F62:[N23:75] F21:180 NXB MOV F29:48 F21:119 NXB SUB F30:74 F30:70 F30:77 NXB CPT F30:71 " F30:70 + ( F30:74 | 4.0 ) " NXB CPT F30:72 " F30:70 + ( 2.0 * ( F30:74 | 4.0 ) ) " NXB CPT F30:73 " F30:70 + ( 3.0 * ( F30:74 | 4.0 ) ) " BND EOR
%   F29:48  PIC461_OUT_FP  "PIC-46-1 Output Value (For HMI Display)" %
%   F30:79  SIC461_SP_FP  "SIC-46-1 PU-46 Flash Evap Circ Pump Speed Setpoint Value (For HMI Display)" %
%   N23:75  PIC461_OUT_PTR  "PIC-46-1 Flash Evap Feed Pres Output Pointer Determines which VFD is controled by FIC" %
%   F21:180  SIC461_AMPS  "PU-46 Current (For HMI Display)" %
%   F21:119  SY461  "SY-46-1 PU-46 Speed (For HMI Display)" %
%   F30:74  SIC461_MAX  "SIC-46-1 PU-46 Flash Evap Circ Pump Speed at 100% Value (For HMI Display)" %
%   F30:70  SIC461_MIN  "SIC-46-1 PU-46 Flash Evap Circ Pump Speed 0% Value (For HMI Display)" %
%   F30:77  SIC461_RANGE  "SIC-46-1 PU-46 Flash Evap Circ Pump Speed Range Value (For HMI Display)" %
%   F30:71  SIC461_25PCNT  "SIC-46-1 PU-46 Flash Evap Circ Pump Speed 25% Value (For HMI Display)" %
%   F30:72  SIC461_50PCNT  "SIC-46-1 PU-46 Flash Evap Circ Pump Speed 50% Value (For HMI Display)" %
%   F30:73  SIC461_75PCNT  "SIC-46-1 PU-46 Flash Evap Circ Pump Speed 75% Value (For HMI Display)" %

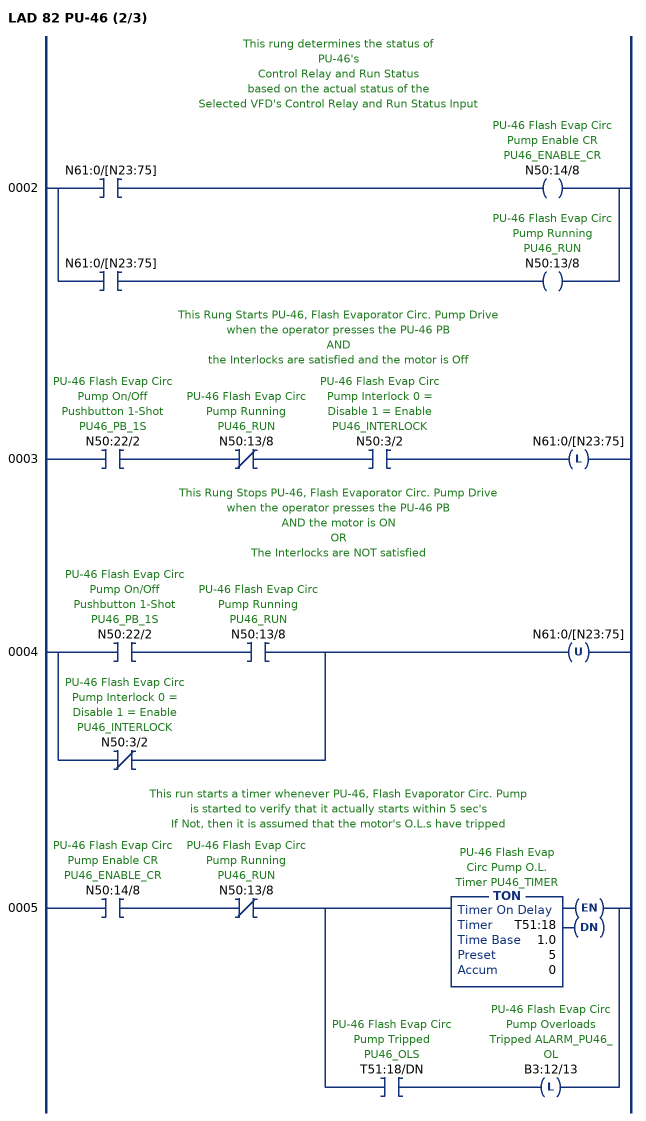
% Rung: 2 %
% This rung determines the status of
% PU-46's
% Control Relay and Run Status
% based on the actual status of the
% Selected VFD's Control Relay and Run Status Input %
SOR BST XIC N61:0/[N23:75] OTE N50:14/8 NXB XIC N61:0/[N23:75] OTE N50:13/8 BND EOR
%   N61:0  VFD_ENABLE_BITS  "These Bits Enable the appropriate VFD" %
%   N23:75  PIC461_OUT_PTR  "PIC-46-1 Flash Evap Feed Pres Output Pointer Determines which VFD is controled by FIC" %
%   N50:14/8  PU46_ENABLE_CR  "PU-46 Flash Evap Circ Pump Enable CR" %
%   N50:13/8  PU46_RUN  "PU-46 Flash Evap Circ Pump Running" %
% Rung: 3 %
% This Rung Starts PU-46, Flash Evaporator Circ. Pump Drive
% when the operator presses the PU-46 PB
% AND
% the Interlocks are satisfied and the motor is Off %
SOR XIC N50:22/2 XIO N50:13/8 XIC N50:3/2 OTL N61:0/[N23:75] EOR
%   N50:22/2  PU46_PB_1S  "PU-46 Flash Evap Circ Pump On/Off Pushbutton 1-Shot" %
%   N50:13/8  PU46_RUN  "PU-46 Flash Evap Circ Pump Running" %
%   N50:3/2  PU46_INTERLOCK  "PU-46 Flash Evap Circ Pump Interlock 0 = Disable 1 = Enable" %
%   N61:0  VFD_ENABLE_BITS  "These Bits Enable the appropriate VFD" %
%   N23:75  PIC461_OUT_PTR  "PIC-46-1 Flash Evap Feed Pres Output Pointer Determines which VFD is controled by FIC" %
% Rung: 4 %
% This Rung Stops PU-46, Flash Evaporator Circ. Pump Drive
% when the operator presses the PU-46 PB
% AND the motor is ON
% OR
% The Interlocks are NOT satisfied %
SOR BST XIC N50:22/2 XIC N50:13/8 NXB XIO N50:3/2 BND OTU N61:0/[N23:75] EOR
%   N50:22/2  PU46_PB_1S  "PU-46 Flash Evap Circ Pump On/Off Pushbutton 1-Shot" %
%   N50:13/8  PU46_RUN  "PU-46 Flash Evap Circ Pump Running" %
%   N50:3/2  PU46_INTERLOCK  "PU-46 Flash Evap Circ Pump Interlock 0 = Disable 1 = Enable" %
%   N61:0  VFD_ENABLE_BITS  "These Bits Enable the appropriate VFD" %
%   N23:75  PIC461_OUT_PTR  "PIC-46-1 Flash Evap Feed Pres Output Pointer Determines which VFD is controled by FIC" %
% Rung: 5 %
% This run starts a timer whenever PU-46, Flash Evaporator Circ. Pump
% is started to verify that it actually starts within 5 sec's
% If Not, then it is assumed that the motor's O.L.s have tripped %
SOR XIC N50:14/8 XIO N50:13/8 BST TON T51:18 1.0 5 0 NXB XIC T51:18/DN OTL B3:12/13 BND EOR
%   N50:14/8  PU46_ENABLE_CR  "PU-46 Flash Evap Circ Pump Enable CR" %
%   N50:13/8  PU46_RUN  "PU-46 Flash Evap Circ Pump Running" %
%   T51:18  PU46_TIMER  "PU-46 Flash Evap Circ Pump O.L. Timer" %
%   T51:18/DN  PU46_OLS  "PU-46 Flash Evap Circ Pump Tripped" %
%   B3:12/13  ALARM_PU46_OL  "PU-46 Flash Evap Circ Pump Overloads Tripped" %

